C07305=1237.701,70.398,-44.996,-178.646,5.352,148.520
C07306=1237.696,70.648,-45.014,-178.643,5.352,148.519
C07307=1237.691,70.897,-45.032,-178.640,5.353,148.519
C07308=1237.686,71.147,-45.049,-178.638,5.353,148.518
C07309=1237.681,71.396,-45.067,-178.635,5.354,148.517
C07310=1237.677,71.645,-45.084,-178.633,5.355,148.517
C07311=1237.671,71.894,-45.102,-178.630,5.355,148.516
C07312=1237.666,72.144,-45.120,-178.628,5.356,148.516
C07313=1237.662,72.393,-45.137,-178.625,5.357,148.515
C07314=1237.656,72.643,-45.155,-178.623,5.357,148.514
C07315=1237.652,72.891,-45.172,-178.620,5.358,148.514
C07316=1237.647,73.141,-45.190,-178.618,5.358,148.513
C07317=1237.642,73.390,-45.208,-178.615,5.358,148.512
C07318=1237.637,73.640,-45.225,-178.613,5.359,148.512
C07319=1237.632,73.889,-45.243,-178.610,5.360,148.511
C07320=1237.627,74.138,-45.261,-178.608,5.360,148.511
C07321=1237.622,74.387,-45.279,-178.605,5.361,148.510
C07322=1237.617,74.637,-45.297,-178.603,5.362,148.509
C07323=1237.613,74.886,-45.314,-178.600,5.362,148.509
C07324=1237.608,75.135,-45.332,-178.597,5.363,148.508
C07325=1237.603,75.384,-45.350,-178.595,5.364,148.508
C07326=1237.599,75.635,-45.368,-178.593,5.364,148.507
C07327=1237.594,75.884,-45.386,-178.590,5.365,148.506
C07328=1237.589,76.133,-45.403,-178.587,5.366,148.506
C07329=1237.584,76.382,-45.421,-178.585,5.366,148.505
C07330=1237.579,76.631,-45.439,-178.582,5.367,148.504
C07331=1237.574,76.880,-45.457,-178.579,5.367,148.504
C07332=1237.569,77.130,-45.475,-178.577,5.368,148.503
C07333=1237.564,77.379,-45.493,-178.575,5.369,148.503
C07334=1237.559,77.629,-45.511,-178.572,5.370,148.502
C07335=1237.555,77.878,-45.528,-178.569,5.370,148.501
C07336=1237.550,78.127,-45.546,-178.567,5.371,148.501
C07337=1237.545,78.376,-45.564,-178.564,5.371,148.500
C07338=1237.541,78.626,-45.582,-178.562,5.372,148.499
C07339=1237.536,78.875,-45.600,-178.559,5.373,148.499
C07340=1237.531,79.125,-45.618,-178.557,5.374,148.498
C07341=1237.526,79.374,-45.636,-178.554,5.374,148.498
C07342=1237.521,79.623,-45.654,-178.552,5.375,148.497
C07343=1237.516,79.872,-45.672,-178.549,5.376,148.496
C07344=1237.511,80.121,-45.690,-178.547,5.376,148.496
C07345=1237.506,80.371,-45.707,-178.544,5.377,148.495
C07346=1237.502,80.620,-45.726,-178.542,5.378,148.494
C07347=1237.497,80.870,-45.744,-178.539,5.378,148.494
C07348=1237.492,81.119,-45.762,-178.536,5.379,148.493
C07349=1237.486,81.368,-45.780,-178.534,5.380,148.493
C07350=1237.481,81.637,-45.800,-178.532,5.380,148.492
C07351=1237.476,81.905,-45.819,-178.529,5.381,148.491
C07352=1237.471,82.173,-45.839,-178.526,5.382,148.491
C07353=1237.466,82.441,-45.858,-178.523,5.383,148.490
C07354=1237.461,82.690,-45.876,-178.520,5.384,148.489
C07355=1237.457,82.940,-45.894,-178.518,5.384,148.489
C07356=1237.452,83.190,-45.912,-178.515,5.385,148.488
C07357=1237.446,83.439,-45.931,-178.513,5.385,148.487
C07358=1237.441,83.688,-45.949,-178.510,5.386,148.487
C07359=1237.436,83.937,-45.967,-178.508,5.387,148.486
C07360=1237.431,84.187,-45.985,-178.505,5.388,148.486
C07361=1237.427,84.436,-46.003,-178.503,5.388,148.485
C07362=1237.422,84.686,-46.021,-178.500,5.389,148.484
C07363=1237.417,84.935,-46.039,-178.497,5.389,148.484
C07364=1237.413,85.183,-46.058,-178.495,5.390,148.483
C07365=1237.408,85.433,-46.076,-178.493,5.391,148.483
C07366=1237.403,85.683,-46.095,-178.490,5.392,148.482
C07367=1237.398,85.932,-46.113,-178.487,5.392,148.481
C07368=1237.393,86.181,-46.131,-178.485,5.393,148.481
C07369=1237.388,86.430,-46.149,-178.483,5.394,148.480
C07370=1237.384,86.680,-46.167,-178.480,5.394,148.480
C07371=1237.379,86.929,-46.186,-178.477,5.395,148.479
C07372=1237.373,87.178,-46.204,-178.475,5.396,148.478
C07373=1237.368,87.427,-46.222,-178.472,5.396,148.478
C07374=1237.364,87.677,-46.241,-178.470,5.397,148.477
C07375=1237.359,87.926,-46.259,-178.467,5.398,148.477
C07376=1237.355,88.175,-46.277,-178.465,5.398,148.476
C07377=1237.349,88.424,-46.296,-178.462,5.399,148.475
C07378=1237.345,88.674,-46.314,-178.460,5.400,148.475
C07379=1237.340,88.923,-46.332,-178.457,5.401,148.474
C07380=1237.335,89.172,-46.351,-178.455,5.401,148.474
C07381=1237.330,89.421,-46.369,-178.452,5.402,148.473
C07382=1237.325,89.671,-46.388,-178.449,5.402,148.472
C07383=1237.320,89.921,-46.406,-178.447,5.403,148.472
C07384=1237.316,90.169,-46.424,-178.445,5.404,148.471
C07385=1237.311,90.419,-46.443,-178.442,5.405,148.471
C07386=1237.306,90.668,-46.461,-178.439,5.405,148.470
C07387=1237.301,90.917,-46.480,-178.437,5.406,148.469
C07388=1237.296,91.166,-46.498,-178.434,5.408,148.469
C07389=1237.291,91.416,-46.517,-178.432,5.408,148.468
C07390=1237.286,91.665,-46.536,-178.429,5.409,148.468
C07391=1237.282,91.914,-46.554,-178.426,5.409,148.467
C07392=1237.277,92.164,-46.572,-178.424,5.410,148.466
C07393=1237.272,92.413,-46.591,-178.422,5.411,148.466
C07394=1237.267,92.662,-46.609,-178.419,5.412,148.465
C07395=1237.263,92.911,-46.628,-178.416,5.412,148.465
C07396=1237.257,93.161,-46.647,-178.414,5.413,148.464
C07397=1237.252,93.410,-46.665,-178.412,5.414,148.463
C07398=1237.248,93.659,-46.684,-178.409,5.414,148.463
C07399=1237.243,93.909,-46.703,-178.406,5.415,148.462
C07400=1237.238,94.157,-46.721,-178.404,5.416,148.461
C07401=1237.234,94.407,-46.740,-178.402,5.417,148.461
C07402=1237.229,94.656,-46.759,-178.399,5.417,148.460
C07403=1237.224,94.905,-46.777,-178.396,5.418,148.460
C07404=1237.219,95.155,-46.795,-178.393,5.419,148.459
C07405=1237.214,95.404,-46.815,-178.391,5.420,148.459
C07406=1237.209,95.653,-46.833,-178.388,5.421,148.458
C07407=1237.204,95.903,-46.852,-178.386,5.422,148.457
C07408=1237.199,96.152,-46.870,-178.383,5.422,148.457
C07409=1237.195,96.401,-46.889,-178.381,5.423,148.456
C07410=1237.190,96.651,-46.908,-178.378,5.424,148.456
C07411=1237.185,96.899,-46.926,-178.376,5.424,148.455
C07412=1237.180,97.149,-46.946,-178.373,5.425,148.454
C07413=1237.175,97.398,-46.964,-178.371,5.426,148.454
C07414=1237.171,97.647,-46.984,-178.368,5.427,148.453
C07415=1237.166,97.897,-47.002,-178.366,5.427,148.453
C07416=1237.161,98.145,-47.020,-178.363,5.428,148.452
C07417=1237.156,98.395,-47.039,-178.361,5.430,148.452
C07418=1237.152,98.644,-47.058,-178.358,5.430,148.451
C07419=1237.147,98.894,-47.078,-178.355,5.431,148.450
C07420=1237.142,99.143,-47.096,-178.353,5.432,148.450
C07421=1237.137,99.392,-47.115,-178.351,5.432,148.449
C07422=1237.132,99.641,-47.133,-178.348,5.433,148.449
C07423=1237.127,99.890,-47.153,-178.345,5.434,148.448
C07424=1237.123,100.140,-47.172,-178.343,5.435,148.448
C07425=1237.117,100.389,-47.190,-178.341,5.435,148.447
C07426=1237.113,100.638,-47.209,-178.338,5.436,148.446
C07427=1237.108,100.887,-47.229,-178.335,5.437,148.446
C07428=1237.104,101.137,-47.247,-178.333,5.438,148.445
C07429=1237.098,101.386,-47.266,-178.330,5.439,148.445
C07430=1237.094,101.635,-47.285,-178.327,5.440,148.444
C07431=1237.089,101.885,-47.304,-178.325,5.440,148.443
C07432=1237.084,102.133,-47.323,-178.323,5.441,148.443
C07433=1237.079,102.383,-47.342,-178.320,5.442,148.442
C07434=1237.075,102.631,-47.361,-178.317,5.442,148.442
C07435=1237.070,102.882,-47.380,-178.315,5.443,148.441
C07436=1237.065,103.130,-47.399,-178.313,5.444,148.440
C07437=1237.060,103.380,-47.418,-178.310,5.445,148.440
C07438=1237.055,103.629,-47.438,-178.307,5.446,148.439
C07439=1237.051,103.878,-47.456,-178.305,5.447,148.439
C07440=1237.045,104.127,-47.475,-178.302,5.448,148.438
C07441=1237.041,104.377,-47.494,-178.300,5.448,148.437
C07442=1237.036,104.625,-47.514,-178.297,5.449,148.437
C07443=1237.031,104.876,-47.532,-178.295,5.450,148.436
C07444=1237.026,105.124,-47.551,-178.292,5.451,148.436
C07445=1237.021,105.374,-47.571,-178.290,5.451,148.435
C07446=1237.017,105.622,-47.590,-178.287,5.453,148.435
C07447=1237.012,105.872,-47.609,-178.284,5.454,148.434
C07448=1237.007,106.121,-47.628,-178.282,5.454,148.433
C07449=1237.003,106.370,-47.648,-178.280,5.455,148.433
C07450=1236.998,106.620,-47.666,-178.277,5.456,148.432
C07451=1236.992,106.869,-47.686,-178.274,5.456,148.432
C07452=1236.988,107.118,-47.705,-178.272,5.457,148.431
C07453=1236.983,107.367,-47.724,-178.270,5.458,148.431
C07454=1236.978,107.636,-47.745,-178.266,5.459,148.430
C07455=1236.973,107.904,-47.766,-178.264,5.460,148.429
C07456=1236.967,108.173,-47.786,-178.261,5.461,148.429
C07457=1236.962,108.442,-47.807,-178.258,5.462,148.428
C07458=1236.958,108.690,-47.826,-178.256,5.463,148.428
C07459=1236.953,108.940,-47.846,-178.253,5.464,148.427
C07460=1236.948,109.189,-47.865,-178.251,5.464,148.426
C07461=1236.943,109.438,-47.885,-178.248,5.465,148.426
C07462=1236.938,109.687,-47.903,-178.246,5.466,148.425
C07463=1236.934,109.936,-47.923,-178.243,5.467,148.425
C07464=1236.929,110.186,-47.943,-178.240,5.468,148.424
C07465=1236.924,110.434,-47.961,-178.238,5.469,148.424
C07466=1236.920,110.684,-47.981,-178.235,5.470,148.423
C07467=1236.914,110.933,-48.000,-178.233,5.470,148.422
C07468=1236.910,111.182,-48.020,-178.231,5.471,148.422
C07469=1236.905,111.432,-48.040,-178.228,5.472,148.421
C07470=1236.900,111.681,-48.058,-178.225,5.473,148.421
C07471=1236.895,111.930,-48.078,-178.223,5.474,148.420
C07472=1236.891,112.180,-48.098,-178.220,5.475,148.420
C07473=1236.885,112.429,-48.117,-178.218,5.476,148.419
C07474=1236.881,112.678,-48.136,-178.215,5.477,148.419
C07475=1236.876,112.926,-48.156,-178.213,5.477,148.418
C07476=1236.872,113.176,-48.176,-178.210,5.479,148.417
C07477=1236.867,113.425,-48.195,-178.208,5.480,148.417
C07478=1236.861,113.674,-48.215,-178.205,5.480,148.416
C07479=1236.857,113.924,-48.234,-178.202,5.481,148.416
C07480=1236.853,114.173,-48.253,-178.200,5.482,148.415
C07481=1236.847,114.422,-48.273,-178.198,5.483,148.415
C07482=1236.843,114.671,-48.292,-178.194,5.484,148.414
C07483=1236.838,114.920,-48.313,-178.192,5.485,148.414
C07484=1236.833,115.169,-48.332,-178.190,5.486,148.413
C07485=1236.828,115.419,-48.352,-178.187,5.486,148.412
C07486=1236.823,115.668,-48.371,-178.185,5.487,148.412
C07487=1236.819,115.917,-48.390,-178.182,5.488,148.411
C07488=1236.814,116.166,-48.410,-178.179,5.489,148.411
C07489=1236.810,116.415,-48.430,-178.177,5.490,148.410
C07490=1236.804,116.664,-48.449,-178.174,5.491,148.410
C07491=1236.799,116.914,-48.469,-178.172,5.492,148.409
C07492=1236.795,117.163,-48.489,-178.170,5.493,148.408
C07493=1236.790,117.412,-48.509,-178.167,5.494,148.408
C07494=1236.785,117.661,-48.528,-178.164,5.495,148.407
C07495=1236.780,117.911,-48.548,-178.162,5.496,148.407
C07496=1236.776,118.160,-48.568,-178.159,5.496,148.406
C07497=1236.770,118.409,-48.588,-178.157,5.497,148.406
C07498=1236.766,118.658,-48.607,-178.154,5.499,148.405
C07499=1236.762,118.907,-48.627,-178.151,5.499,148.405
C07500=1236.757,119.156,-48.647,-178.149,5.500,148.404
C07501=1236.752,119.405,-48.666,-178.147,5.501,148.403
C07502=1236.747,119.654,-48.686,-178.144,5.502,148.403
C07503=1236.743,119.904,-48.706,-178.142,5.503,148.402
C07504=1236.738,120.153,-48.726,-178.139,5.504,148.402
C07505=1236.733,120.402,-48.746,-178.136,5.505,148.401
C07506=1236.728,120.651,-48.765,-178.134,5.506,148.401
C07507=1236.723,120.901,-48.785,-178.131,5.506,148.400
C07508=1236.719,121.150,-48.805,-178.128,5.508,148.399
C07509=1236.714,121.399,-48.825,-178.126,5.509,148.399
C07510=1236.709,121.647,-48.845,-178.123,5.509,148.398
C07511=1236.704,121.897,-48.865,-178.121,5.510,148.398
C07512=1236.700,122.147,-48.884,-178.119,5.511,148.397
C07513=1236.695,122.396,-48.905,-178.116,5.513,148.397
C07514=1236.689,122.645,-48.925,-178.113,5.513,148.396
C07515=1236.685,122.894,-48.945,-178.111,5.514,148.396
C07516=1236.680,123.143,-48.965,-178.109,5.515,148.395
C07517=1236.676,123.392,-48.985,-178.106,5.516,148.395
C07518=1236.671,123.642,-49.005,-178.103,5.517,148.394
C07519=1236.666,123.890,-49.025,-178.101,5.518,148.394
C07520=1236.661,124.140,-49.044,-178.098,5.519,148.393
C07521=1236.657,124.389,-49.065,-178.096,5.519,148.392
C07522=1236.652,124.638,-49.084,-178.093,5.521,148.392
C07523=1236.647,124.887,-49.105,-178.090,5.522,148.391
C07524=1236.643,125.137,-49.124,-178.088,5.523,148.391
C07525=1236.638,125.385,-49.144,-178.086,5.524,148.390
C07526=1236.632,125.635,-49.165,-178.083,5.524,148.390
C07527=1236.628,125.884,-49.185,-178.080,5.526,148.389
C07528=1236.623,126.133,-49.205,-178.078,5.527,148.389
C07529=1236.619,126.382,-49.225,-178.076,5.528,148.388
C07530=1236.614,126.631,-49.245,-178.073,5.528,148.388
C07531=1236.609,126.880,-49.265,-178.070,5.530,148.387
C07532=1236.604,127.129,-49.285,-178.068,5.531,148.387
C07533=1236.599,127.378,-49.306,-178.065,5.531,148.386
C07534=1236.594,127.628,-49.326,-178.063,5.532,148.386
C07535=1236.590,127.877,-49.346,-178.060,5.534,148.385
C07536=1236.585,128.126,-49.366,-178.057,5.534,148.384
C07537=1236.581,128.375,-49.386,-178.055,5.535,148.384
C07538=1236.576,128.624,-49.406,-178.053,5.536,148.383
C07539=1236.571,128.874,-49.427,-178.050,5.538,148.383
C07540=1236.566,129.122,-49.447,-178.047,5.539,148.382
C07541=1236.561,129.371,-49.467,-178.045,5.539,148.382
C07542=1236.557,129.620,-49.487,-178.043,5.540,148.381
C07543=1236.552,129.870,-49.508,-178.039,5.542,148.381
C07544=1236.547,130.119,-49.528,-178.037,5.543,148.380
C07545=1236.543,130.368,-49.548,-178.035,5.543,148.380
C07546=1236.538,130.618,-49.568,-178.033,5.544,148.379
C07547=1236.533,130.867,-49.588,-178.029,5.546,148.379
C07548=1236.528,131.116,-49.609,-178.027,5.546,148.378
C07549=1236.524,131.365,-49.630,-178.025,5.547,148.377
C07550=1236.519,131.614,-49.650,-178.022,5.548,148.377
C07551=1236.514,131.864,-49.670,-178.019,5.550,148.376
C07552=1236.509,132.112,-49.690,-178.017,5.551,148.376
C07553=1236.504,132.361,-49.711,-178.015,5.552,148.375
C07554=1236.500,132.610,-49.731,-178.012,5.553,148.375
C07555=1236.495,132.859,-49.752,-178.009,5.554,148.374
C07556=1236.490,133.109,-49.772,-178.007,5.555,148.374
C07557=1236.486,133.357,-49.792,-178.004,5.555,148.373
C07558=1236.480,133.626,-49.815,-178.001,5.557,148.373
C07559=1236.475,133.896,-49.837,-177.999,5.558,148.372
C07560=1236.470,134.164,-49.859,-177.996,5.559,148.372
C07561=1236.465,134.432,-49.881,-177.993,5.560,148.371
C07562=1236.460,134.681,-49.902,-177.991,5.561,148.370
C07563=1236.455,134.931,-49.921,-177.988,5.562,148.370
C07564=1236.451,135.180,-49.942,-177.986,5.563,148.369
C07565=1236.446,135.429,-49.963,-177.983,5.564,148.369
C07566=1236.441,135.678,-49.983,-177.980,5.565,148.368
C07567=1236.436,135.927,-50.004,-177.978,5.566,148.368
C07568=1236.432,136.176,-50.024,-177.975,5.567,148.367
C07569=1236.427,136.425,-50.045,-177.973,5.568,148.367
C07570=1236.422,136.674,-50.066,-177.970,5.570,148.366
C07571=1236.418,136.923,-50.086,-177.968,5.571,148.366
C07572=1236.413,137.172,-50.107,-177.965,5.571,148.365
C07573=1236.408,137.421,-50.127,-177.963,5.573,148.365
C07574=1236.404,137.670,-50.148,-177.960,5.574,148.364
C07575=1236.398,137.920,-50.169,-177.958,5.575,148.364
C07576=1236.395,138.169,-50.190,-177.955,5.576,148.363
C07577=1236.389,138.419,-50.211,-177.952,5.577,148.363
C07578=1236.385,138.668,-50.231,-177.950,5.578,148.362
C07579=1236.380,138.917,-50.252,-177.948,5.578,148.361
C07580=1236.375,139.166,-50.272,-177.945,5.580,148.361
C07581=1236.370,139.415,-50.293,-177.942,5.581,148.360
C07582=1236.366,139.664,-50.314,-177.940,5.582,148.360
C07583=1236.361,139.913,-50.335,-177.937,5.583,148.359
C07584=1236.356,140.162,-50.356,-177.935,5.584,148.359
C07585=1236.351,140.411,-50.377,-177.932,5.585,148.358
C07586=1236.347,140.660,-50.397,-177.930,5.587,148.358
C07587=1236.342,140.909,-50.418,-177.927,5.588,148.357
C07588=1236.337,141.158,-50.438,-177.925,5.589,148.357
C07589=1236.332,141.407,-50.459,-177.922,5.590,148.356
C07590=1236.328,141.656,-50.480,-177.920,5.591,148.356
C07591=1236.323,141.906,-50.501,-177.917,5.592,148.355
C07592=1236.319,142.154,-50.522,-177.914,5.593,148.355
C07593=1236.314,142.404,-50.543,-177.912,5.594,148.354
C07594=1236.309,142.653,-50.563,-177.910,5.595,148.354
C07595=1236.304,142.902,-50.584,-177.907,5.597,148.353
C07596=1236.300,143.151,-50.605,-177.904,5.598,148.353
C07597=1236.295,143.399,-50.626,-177.902,5.598,148.352
C07598=1236.290,143.649,-50.647,-177.899,5.600,148.352
C07599=1236.286,143.898,-50.668,-177.897,5.601,148.351
C07600=1236.281,144.148,-50.689,-177.894,5.601,148.351
C07601=1236.277,144.396,-50.710,-177.891,5.603,148.350
C07602=1236.271,144.645,-50.731,-177.889,5.604,148.350
C07603=1236.266,144.894,-50.752,-177.887,5.605,148.349
C07604=1236.262,145.143,-50.772,-177.883,5.606,148.349
C07605=1236.257,145.392,-50.794,-177.881,5.607,148.348
C07606=1236.253,145.642,-50.815,-177.879,5.608,148.348
C07607=1236.248,145.891,-50.836,-177.876,5.610,148.347
C07608=1236.243,146.140,-50.858,-177.874,5.611,148.347
C07609=1236.239,146.389,-50.878,-177.871,5.612,148.346
C07610=1236.233,146.638,-50.899,-177.868,5.613,148.346
C07611=1236.229,146.886,-50.921,-177.866,5.614,148.345
C07612=1236.225,147.136,-50.941,-177.864,5.615,148.345
C07613=1236.220,147.385,-50.962,-177.861,5.616,148.344
C07614=1236.215,147.634,-50.984,-177.859,5.617,148.344
C07615=1236.210,147.883,-51.004,-177.856,5.618,148.343
C07616=1236.205,148.132,-51.026,-177.854,5.620,148.343
C07617=1236.201,148.382,-51.047,-177.851,5.621,148.342
C07618=1236.196,148.631,-51.068,-177.848,5.622,148.342
C07619=1236.191,148.879,-51.089,-177.846,5.623,148.341
C07620=1236.186,149.128,-51.110,-177.844,5.624,148.341
C07621=1236.182,149.378,-51.132,-177.840,5.626,148.340
C07622=1236.178,149.627,-51.153,-177.838,5.627,148.340
C07623=1236.173,149.875,-51.174,-177.836,5.627,148.339
C07624=1236.168,150.125,-51.195,-177.833,5.629,148.339
C07625=1236.163,150.373,-51.217,-177.830,5.630,148.338
C07626=1236.159,150.623,-51.238,-177.828,5.632,148.338
C07627=1236.154,150.872,-51.260,-177.825,5.632,148.337
C07628=1236.149,151.121,-51.281,-177.823,5.633,148.337
C07629=1236.144,151.369,-51.302,-177.820,5.635,148.336
C07630=1236.140,151.619,-51.323,-177.818,5.636,148.336
C07631=1236.135,151.868,-51.345,-177.815,5.636,148.335
C07632=1236.130,152.117,-51.366,-177.813,5.638,148.335
C07633=1236.125,152.366,-51.387,-177.811,5.639,148.334
C07634=1236.121,152.616,-51.409,-177.807,5.641,148.334
C07635=1236.116,152.864,-51.430,-177.805,5.642,148.333
C07636=1236.111,153.113,-51.451,-177.803,5.642,148.333
C07637=1236.107,153.363,-51.473,-177.800,5.644,148.332
C07638=1236.102,153.611,-51.494,-177.797,5.645,148.332
C07639=1236.097,153.860,-51.515,-177.795,5.647,148.332
C07640=1236.092,154.109,-51.537,-177.792,5.647,148.331
C07641=1236.088,154.359,-51.558,-177.790,5.648,148.330
C07642=1236.083,154.607,-51.579,-177.787,5.650,148.330
C07643=1236.079,154.856,-51.601,-177.785,5.651,148.329
C07644=1236.074,155.106,-51.622,-177.782,5.653,148.329
C07645=1236.069,155.355,-51.644,-177.780,5.653,148.328
C07646=1236.064,155.603,-51.666,-177.777,5.654,148.328
C07647=1236.060,155.853,-51.687,-177.774,5.656,148.328
C07648=1236.055,156.102,-51.709,-177.772,5.657,148.327
C07649=1236.050,156.350,-51.731,-177.769,5.658,148.327
C07650=1236.046,156.600,-51.753,-177.767,5.659,148.326
C07651=1236.041,156.849,-51.773,-177.765,5.660,148.326
C07652=1236.036,157.097,-51.795,-177.762,5.662,148.325
C07653=1236.032,157.347,-51.817,-177.760,5.663,148.325
C07654=1236.027,157.595,-51.838,-177.756,5.664,148.324
C07655=1236.022,157.845,-51.859,-177.754,5.665,148.324
C07656=1236.018,158.094,-51.881,-177.752,5.666,148.323
C07657=1236.013,158.343,-51.903,-177.749,5.668,148.323
C07658=1236.009,158.592,-51.925,-177.747,5.669,148.322
C07659=1236.004,158.841,-51.947,-177.744,5.670,148.322
C07660=1235.999,159.090,-51.968,-177.742,5.671,148.321
C07661=1235.994,159.339,-51.990,-177.739,5.673,148.321
C07662=1235.989,159.608,-52.014,-177.737,5.674,148.320
C07663=1235.984,159.877,-52.037,-177.733,5.675,148.320
C07664=1235.979,160.146,-52.060,-177.731,5.676,148.319
C07665=1235.974,160.415,-52.084,-177.728,5.678,148.319
C07666=1235.969,160.664,-52.106,-177.725,5.679,148.318
C07667=1235.964,160.914,-52.127,-177.723,5.680,148.318
C07668=1235.959,161.162,-52.149,-177.721,5.681,148.317
C07669=1235.955,161.412,-52.171,-177.718,5.683,148.317
C07670=1235.950,161.660,-52.193,-177.716,5.684,148.316
C07671=1235.946,161.910,-52.215,-177.712,5.685,148.316
C07672=1235.941,162.158,-52.236,-177.710,5.686,148.315
C07673=1235.936,162.407,-52.258,-177.708,5.688,148.315
C07674=1235.932,162.656,-52.280,-177.705,5.689,148.315
C07675=1235.927,162.905,-52.302,-177.702,5.691,148.314
C07676=1235.923,163.154,-52.324,-177.700,5.691,148.314
C07677=1235.918,163.403,-52.345,-177.698,5.692,148.313
C07678=1235.913,163.653,-52.368,-177.695,5.694,148.313
C07679=1235.908,163.901,-52.390,-177.692,5.695,148.312
C07680=1235.904,164.151,-52.412,-177.690,5.697,148.312
C07681=1235.899,164.399,-52.433,-177.687,5.697,148.311
C07682=1235.895,164.649,-52.455,-177.685,5.699,148.311
C07683=1235.890,164.897,-52.477,-177.682,5.700,148.310
C07684=1235.886,165.147,-52.499,-177.679,5.702,148.310
C07685=1235.881,165.395,-52.521,-177.677,5.703,148.309
C07686=1235.876,165.645,-52.544,-177.674,5.704,148.309
C07687=1235.871,165.893,-52.565,-177.672,5.705,148.308
C07688=1235.867,166.143,-52.587,-177.669,5.707,148.308
C07689=1235.862,166.391,-52.609,-177.667,5.708,148.307
C07690=1235.858,166.640,-52.632,-177.665,5.709,148.307
C07691=1235.853,166.889,-52.653,-177.662,5.711,148.307
C07692=1235.848,167.138,-52.676,-177.659,5.711,148.306
C07693=1235.843,167.387,-52.698,-177.657,5.713,148.306
C07694=1235.839,167.636,-52.720,-177.654,5.714,148.305
C07695=1235.834,167.885,-52.741,-177.652,5.716,148.305
C07696=1235.830,168.134,-52.764,-177.649,5.717,148.304
C07697=1235.824,168.383,-52.786,-177.646,5.718,148.304
C07698=1235.820,168.632,-52.809,-177.644,5.719,148.303
C07699=1235.815,168.881,-52.830,-177.642,5.721,148.303
C07700=1235.811,169.130,-52.852,-177.639,5.722,148.302
C07701=1235.805,169.379,-52.875,-177.636,5.724,148.302
C07702=1235.801,169.628,-52.897,-177.634,5.725,148.302
C07703=1235.796,169.876,-52.919,-177.631,5.726,148.301
C07704=1235.792,170.126,-52.941,-177.629,5.727,148.301
C07705=1235.787,170.375,-52.964,-177.626,5.729,148.300
C07706=1235.783,170.623,-52.986,-177.624,5.730,148.300
C07707=1235.778,170.873,-53.008,-177.621,5.732,148.299
C07708=1235.773,171.122,-53.030,-177.619,5.732,148.299
C07709=1235.768,171.371,-53.052,-177.616,5.734,148.298
C07710=1235.764,171.619,-53.075,-177.614,5.735,148.298
C07711=1235.760,171.868,-53.097,-177.611,5.737,148.297
C07712=1235.755,172.118,-53.120,-177.609,5.738,148.297
C07713=1235.750,172.366,-53.142,-177.606,5.739,148.297
C07714=1235.746,172.615,-53.164,-177.603,5.740,148.296
C07715=1235.740,172.864,-53.186,-177.601,5.742,148.296
C07716=1235.736,173.113,-53.209,-177.599,5.743,148.295
C07717=1235.731,173.363,-53.232,-177.595,5.744,148.295
C07718=1235.727,173.611,-53.254,-177.593,5.745,148.294
C07719=1235.722,173.860,-53.276,-177.591,5.747,148.294
C07720=1235.717,174.110,-53.299,-177.588,5.748,148.293
C07721=1235.713,174.358,-53.321,-177.585,5.750,148.293
C07722=1235.709,174.607,-53.343,-177.583,5.751,148.293
C07723=1235.703,174.855,-53.366,-177.580,5.752,148.292
C07724=1235.699,175.105,-53.388,-177.578,5.753,148.292
C07725=1235.694,175.354,-53.411,-177.576,5.755,148.291
C07726=1235.689,175.602,-53.433,-177.573,5.756,148.291
C07727=1235.685,175.852,-53.455,-177.570,5.758,148.290
C07728=1235.680,176.101,-53.479,-177.568,5.760,148.290
C07729=1235.676,176.349,-53.500,-177.565,5.760,148.289
C07730=1235.671,176.598,-53.524,-177.562,5.762,148.289
C07731=1235.667,176.848,-53.546,-177.560,5.763,148.289
C07732=1235.661,177.096,-53.569,-177.557,5.765,148.288
C07733=1235.657,177.346,-53.591,-177.555,5.766,148.288
C07734=1235.652,177.595,-53.614,-177.552,5.768,148.287
C07735=1235.648,177.843,-53.637,-177.550,5.769,148.287
C07736=1235.643,178.092,-53.659,-177.547,5.770,148.286
C07737=1235.639,178.341,-53.682,-177.545,5.771,148.286
C07738=1235.634,178.591,-53.705,-177.542,5.773,148.286
C07739=1235.629,178.839,-53.727,-177.540,5.774,148.285
C07740=1235.624,179.088,-53.750,-177.537,5.775,148.285
C07741=1235.620,179.337,-53.772,-177.535,5.777,148.284
C07742=1235.615,179.585,-53.795,-177.532,5.778,148.284
C07743=1235.611,179.835,-53.817,-177.529,5.780,148.283
C07744=1235.606,180.084,-53.841,-177.527,5.781,148.283
C07745=1235.602,180.332,-53.864,-177.524,5.782,148.282
C07746=1235.596,180.581,-53.886,-177.522,5.783,148.282
C07747=1235.592,180.830,-53.909,-177.519,5.785,148.282
C07748=1235.588,181.079,-53.932,-177.517,5.786,148.281
C07749=1235.583,181.329,-53.955,-177.514,5.788,148.281
C07750=1235.578,181.577,-53.977,-177.512,5.790,148.280
C07751=1235.574,181.826,-54.000,-177.509,5.791,148.280
C07752=1235.569,182.075,-54.022,-177.506,5.792,148.279
C07753=1235.565,182.324,-54.046,-177.504,5.793,148.279
C07754=1235.560,182.572,-54.068,-177.502,5.795,148.279
C07755=1235.555,182.821,-54.092,-177.500,5.796,148.278
C07756=1235.550,183.071,-54.114,-177.496,5.798,148.278
C07757=1235.546,183.320,-54.137,-177.494,5.799,148.277
C07758=1235.542,183.569,-54.160,-177.492,5.800,148.277
C07759=1235.536,183.817,-54.183,-177.489,5.802,148.276
C07760=1235.532,184.066,-54.206,-177.486,5.803,148.276
C07761=1235.527,184.315,-54.229,-177.484,5.805,148.276
C07762=1235.523,184.564,-54.252,-177.481,5.807,148.275
C07763=1235.519,184.813,-54.275,-177.479,5.807,148.275
C07764=1235.513,185.061,-54.298,-177.476,5.809,148.274
C07765=1235.509,185.310,-54.321,-177.474,5.810,148.274
C07766=1235.504,185.580,-54.346,-177.471,5.812,148.273
C07767=1235.499,185.850,-54.371,-177.468,5.814,148.273
C07768=1235.494,186.120,-54.396,-177.465,5.815,148.272
C07769=1235.489,186.390,-54.421,-177.462,5.817,148.272
C07770=1235.484,186.638,-54.444,-177.460,5.818,148.272
C07771=1235.479,186.887,-54.467,-177.458,5.820,148.271
C07772=1235.476,187.136,-54.490,-177.455,5.821,148.271
C07773=1235.471,187.385,-54.513,-177.452,5.822,148.270
C07774=1235.466,187.634,-54.536,-177.450,5.824,148.270
C07775=1235.461,187.883,-54.560,-177.447,5.825,148.270
C07776=1235.457,188.132,-54.582,-177.445,5.827,148.269
C07777=1235.452,188.380,-54.605,-177.442,5.828,148.269
C07778=1235.447,188.629,-54.629,-177.440,5.830,148.268
C07779=1235.443,188.878,-54.652,-177.437,5.832,148.268
C07780=1235.439,189.127,-54.675,-177.435,5.832,148.267
C07781=1235.434,189.376,-54.698,-177.432,5.834,148.267
C07782=1235.429,189.625,-54.722,-177.430,5.835,148.267
C07783=1235.425,189.874,-54.745,-177.427,5.837,148.266
C07784=1235.420,190.123,-54.768,-177.424,5.838,148.266
C07785=1235.415,190.372,-54.792,-177.422,5.839,148.265
C07786=1235.411,190.620,-54.814,-177.419,5.841,148.265
C07787=1235.406,190.869,-54.838,-177.417,5.843,148.265
C07788=1235.401,191.118,-54.861,-177.414,5.844,148.264
C07789=1235.397,191.367,-54.884,-177.412,5.846,148.264
C07790=1235.392,191.616,-54.908,-177.409,5.847,148.263
C07791=1235.387,191.865,-54.931,-177.407,5.849,148.263
C07792=1235.383,192.114,-54.954,-177.404,5.850,148.263
C07793=1235.379,192.362,-54.978,-177.402,5.851,148.262
C07794=1235.374,192.611,-55.001,-177.399,5.853,148.262
C07795=1235.369,192.860,-55.025,-177.396,5.855,148.261
C07796=1235.365,193.109,-55.048,-177.394,5.856,148.261
C07797=1235.360,193.358,-55.071,-177.391,5.857,148.261
C07798=1235.355,193.607,-55.095,-177.389,5.858,148.260
C07799=1235.351,193.856,-55.119,-177.386,5.860,148.260
C07800=1235.346,194.105,-55.142,-177.384,5.862,148.259
C07801=1235.342,194.354,-55.165,-177.381,5.863,148.259
C07802=1235.337,194.603,-55.189,-177.379,5.865,148.258
C07803=1235.332,194.851,-55.211,-177.376,5.867,148.258
C07804=1235.328,195.099,-55.235,-177.374,5.868,148.258
C07805=1235.323,195.348,-55.259,-177.371,5.869,148.257
C07806=1235.319,195.597,-55.282,-177.368,5.871,148.257
C07807=1235.314,195.846,-55.305,-177.366,5.872,148.256
C07808=1235.309,196.095,-55.329,-177.363,5.874,148.256
C07809=1235.305,196.344,-55.353,-177.361,5.876,148.256
C07810=1235.300,196.593,-55.376,-177.359,5.877,148.255
C07811=1235.296,196.841,-55.400,-177.355,5.878,148.255
C07812=1235.291,197.090,-55.424,-177.353,5.880,148.255
C07813=1235.287,197.340,-55.447,-177.351,5.881,148.254
C07814=1235.282,197.588,-55.471,-177.348,5.883,148.254
C07815=1235.278,197.837,-55.495,-177.345,5.885,148.253
C07816=1235.273,198.086,-55.518,-177.343,5.886,148.253
C07817=1235.269,198.335,-55.542,-177.340,5.887,148.253
C07818=1235.264,198.584,-55.565,-177.338,5.889,148.252
C07819=1235.260,198.832,-55.590,-177.336,5.890,148.252
C07820=1235.255,199.081,-55.613,-177.333,5.892,148.251
C07821=1235.249,199.331,-55.637,-177.330,5.894,148.251
C07822=1235.245,199.579,-55.661,-177.328,5.895,148.251
C07823=1235.240,199.828,-55.684,-177.325,5.897,148.250
C07824=1235.236,200.077,-55.708,-177.322,5.898,148.250
C07825=1235.231,200.326,-55.732,-177.320,5.900,148.249
C07826=1235.227,200.574,-55.756,-177.318,5.901,148.249
C07827=1235.222,200.823,-55.779,-177.315,5.903,148.249
C07828=1235.218,201.071,-55.803,-177.312,5.905,148.248
C07829=1235.213,201.320,-55.827,-177.310,5.906,148.248
C07830=1235.209,201.570,-55.851,-177.307,5.908,148.248
C07831=1235.204,201.819,-55.875,-177.305,5.910,148.247
C07832=1235.199,202.067,-55.899,-177.303,5.911,148.247
C07833=1235.195,202.316,-55.922,-177.299,5.912,148.246
C07834=1235.190,202.565,-55.946,-177.297,5.914,148.246
C07835=1235.186,202.814,-55.970,-177.295,5.915,148.246
C07836=1235.181,203.062,-55.994,-177.292,5.917,148.245
C07837=1235.177,203.311,-56.018,-177.289,5.919,148.245
C07838=1235.171,203.560,-56.042,-177.287,5.921,148.245
C07839=1235.168,203.809,-56.066,-177.284,5.921,148.244
C07840=1235.163,204.058,-56.090,-177.282,5.923,148.244
C07841=1235.159,204.307,-56.114,-177.279,5.925,148.243
C07842=1235.154,204.555,-56.138,-177.277,5.926,148.243
C07843=1235.149,204.804,-56.162,-177.274,5.928,148.243
C07844=1235.144,205.053,-56.186,-177.272,5.930,148.242
C07845=1235.140,205.302,-56.210,-177.269,5.932,148.242
C07846=1235.136,205.551,-56.234,-177.266,5.932,148.241
C07847=1235.131,205.800,-56.258,-177.264,5.934,148.241
C07848=1235.126,206.048,-56.282,-177.261,5.936,148.241
C07849=1235.122,206.297,-56.306,-177.259,5.937,148.240
C07850=1235.117,206.545,-56.330,-177.257,5.939,148.240
C07851=1235.113,206.795,-56.355,-177.254,5.941,148.240
C07852=1235.108,207.043,-56.379,-177.251,5.943,148.239
C07853=1235.104,207.292,-56.402,-177.249,5.943,148.239
C07854=1235.099,207.541,-56.426,-177.246,5.945,148.238
C07855=1235.094,207.789,-56.451,-177.243,5.947,148.238
C07856=1235.090,208.039,-56.476,-177.241,5.949,148.238
C07857=1235.086,208.288,-56.499,-177.239,5.950,148.237
C07858=1235.080,208.536,-56.524,-177.236,5.952,148.237
C07859=1235.076,208.785,-56.548,-177.233,5.954,148.237
C07860=1235.072,209.033,-56.572,-177.231,5.955,148.236
C07861=1235.067,209.283,-56.597,-177.228,5.956,148.236
C07862=1235.063,209.531,-56.621,-177.226,5.958,148.235
C07863=1235.058,209.780,-56.644,-177.223,5.960,148.235
C07864=1235.053,210.029,-56.669,-177.221,5.961,148.235
C07865=1235.049,210.278,-56.693,-177.218,5.963,148.234
C07866=1235.044,210.527,-56.718,-177.216,5.965,148.234
C07867=1235.040,210.775,-56.742,-177.213,5.967,148.234
C07868=1235.035,211.023,-56.766,-177.211,5.968,148.233
C07869=1235.031,211.273,-56.791,-177.208,5.969,148.233
C07870=1235.025,211.544,-56.817,-177.205,5.971,148.232
C07871=1235.021,211.813,-56.843,-177.203,5.973,148.232
C07872=1235.016,212.084,-56.870,-177.200,5.975,148.232
C07873=1235.010,212.354,-56.897,-177.197,5.976,148.231
C07874=1235.007,212.603,-56.921,-177.194,5.978,148.231
C07875=1235.002,212.852,-56.946,-177.192,5.980,148.230
C07876=1234.997,213.100,-56.970,-177.189,5.982,148.230
C07877=1234.993,213.349,-56.995,-177.187,5.983,148.230
C07878=1234.988,213.598,-57.019,-177.184,5.985,148.229
C07879=1234.983,213.847,-57.044,-177.182,5.987,148.229
C07880=1234.979,214.096,-57.068,-177.179,5.989,148.229
C07881=1234.974,214.344,-57.093,-177.177,5.990,148.228
C07882=1234.970,214.593,-57.117,-177.174,5.991,148.228
C07883=1234.965,214.842,-57.142,-177.171,5.993,148.228
C07884=1234.961,215.091,-57.166,-177.169,5.995,148.227
C07885=1234.956,215.339,-57.191,-177.166,5.997,148.227
C07886=1234.952,215.589,-57.215,-177.164,5.998,148.227
C07887=1234.947,215.837,-57.240,-177.161,6.000,148.226
C07888=1234.942,216.086,-57.264,-177.159,6.002,148.226
C07889=1234.938,216.334,-57.290,-177.156,6.004,148.226
C07890=1234.934,216.583,-57.314,-177.153,6.005,148.225
C07891=1234.929,216.832,-57.338,-177.151,6.006,148.225
C07892=1234.925,217.081,-57.363,-177.149,6.008,148.225
C07893=1234.920,217.329,-57.387,-177.146,6.010,148.224
C07894=1234.915,217.578,-57.412,-177.143,6.012,148.224
C07895=1234.911,217.827,-57.437,-177.140,6.014,148.223
C07896=1234.906,218.075,-57.462,-177.138,6.015,148.223
C07897=1234.902,218.324,-57.486,-177.136,6.016,148.223
C07898=1234.897,218.573,-57.511,-177.133,6.018,148.222
C07899=1234.892,218.822,-57.536,-177.130,6.020,148.222
C07900=1234.888,219.070,-57.561,-177.128,6.022,148.222
C07901=1234.883,219.319,-57.586,-177.126,6.023,148.221
C07902=1234.879,219.568,-57.610,-177.123,6.025,148.221
C07903=1234.875,219.816,-57.635,-177.120,6.027,148.221
C07904=1234.870,220.065,-57.660,-177.118,6.029,148.220
C07905=1234.866,220.314,-57.684,-177.115,6.031,148.220
C07906=1234.861,220.563,-57.709,-177.113,6.032,148.220
C07907=1234.856,220.812,-57.735,-177.111,6.034,148.219
C07908=1234.852,221.060,-57.759,-177.108,6.035,148.219
C07909=1234.847,221.310,-57.784,-177.105,6.037,148.219
C07910=1234.843,221.558,-57.809,-177.103,6.039,148.218
C07911=1234.838,221.806,-57.833,-177.101,6.040,148.218
C07912=1234.834,222.055,-57.859,-177.097,6.042,148.217
C07913=1234.829,222.304,-57.884,-177.095,6.044,148.217
C07914=1234.825,222.553,-57.908,-177.092,6.046,148.217
C07915=1234.820,222.801,-57.934,-177.090,6.047,148.216
C07916=1234.816,223.050,-57.959,-177.088,6.048,148.216
C07917=1234.811,223.298,-57.984,-177.085,6.050,148.216
C07918=1234.807,223.547,-58.009,-177.082,6.052,148.215
C07919=1234.802,223.796,-58.033,-177.080,6.054,148.215
C07920=1234.798,224.045,-58.059,-177.077,6.056,148.215
C07921=1234.793,224.294,-58.084,-177.074,6.058,148.214
C07922=1234.789,224.542,-58.109,-177.072,6.059,148.214
C07923=1234.784,224.791,-58.133,-177.070,6.061,148.214
C07924=1234.780,225.040,-58.159,-177.067,6.063,148.213
C07925=1234.775,225.288,-58.184,-177.065,6.064,148.213
C07926=1234.770,225.537,-58.210,-177.062,6.066,148.213
C07927=1234.766,225.786,-58.234,-177.059,6.068,148.212
C07928=1234.762,226.034,-58.259,-177.057,6.069,148.212
C07929=1234.757,226.283,-58.284,-177.055,6.071,148.212
C07930=1234.752,226.532,-58.310,-177.052,6.073,148.211
C07931=1234.748,226.780,-58.335,-177.049,6.075,148.211
C07932=1234.743,227.030,-58.360,-177.047,6.077,148.211
C07933=1234.739,227.277,-58.385,-177.044,6.079,148.210
C07934=1234.734,227.527,-58.410,-177.042,6.080,148.210
C07935=1234.730,227.775,-58.436,-177.039,6.082,148.210
C07936=1234.725,228.024,-58.461,-177.037,6.083,148.209
C07937=1234.720,228.272,-58.486,-177.034,6.085,148.209
C07938=1234.716,228.521,-58.512,-177.032,6.087,148.209
C07939=1234.712,228.770,-58.537,-177.029,6.089,148.208
C07940=1234.707,229.019,-58.562,-177.027,6.090,148.208
C07941=1234.703,229.267,-58.587,-177.024,6.092,148.208
C07942=1234.698,229.515,-58.613,-177.022,6.094,148.207
C07943=1234.694,229.765,-58.638,-177.019,6.096,148.207
C07944=1234.690,230.014,-58.663,-177.016,6.098,148.207
C07945=1234.685,230.262,-58.689,-177.014,6.100,148.207
C07946=1234.681,230.510,-58.715,-177.012,6.101,148.206
C07947=1234.675,230.759,-58.739,-177.010,6.103,148.206
C07948=1234.671,231.008,-58.765,-177.007,6.105,148.206
C07949=1234.667,231.257,-58.791,-177.004,6.107,148.205
C07950=1234.662,231.505,-58.816,-177.002,6.108,148.205
C07951=1234.658,231.754,-58.841,-176.999,6.110,148.205
C07952=1234.653,232.002,-58.867,-176.997,6.112,148.204
C07953=1234.649,232.251,-58.892,-176.994,6.113,148.204
C07954=1234.644,232.500,-58.918,-176.992,6.115,148.204
C07955=1234.640,232.748,-58.943,-176.989,6.117,148.203
C07956=1234.635,232.998,-58.968,-176.987,6.119,148.203
C07957=1234.631,233.246,-58.994,-176.984,6.121,148.203
C07958=1234.626,233.494,-59.020,-176.981,6.123,148.203
C07959=1234.622,233.743,-59.045,-176.979,6.124,148.202
C07960=1234.617,233.992,-59.071,-176.977,6.126,148.202
C07961=1234.613,234.240,-59.096,-176.974,6.127,148.202
C07962=1234.608,234.489,-59.122,-176.971,6.129,148.201
C07963=1234.604,234.738,-59.148,-176.969,6.131,148.201
C07964=1234.599,234.986,-59.173,-176.966,6.133,148.201
C07965=1234.595,235.235,-59.198,-176.964,6.135,148.200
C07966=1234.591,235.484,-59.224,-176.961,6.137,148.200
C07967=1234.585,235.733,-59.250,-176.959,6.139,148.200
C07968=1234.581,235.981,-59.276,-176.957,6.140,148.199
C07969=1234.577,236.230,-59.302,-176.954,6.142,148.199
C07970=1234.572,236.478,-59.327,-176.952,6.144,148.199
C07971=1234.568,236.727,-59.353,-176.949,6.146,148.199
C07972=1234.563,236.976,-59.379,-176.946,6.148,148.198
C07973=1234.559,237.224,-59.404,-176.944,6.149,148.198
C07974=1234.554,237.495,-59.433,-176.941,6.151,148.198
C07975=1234.549,237.767,-59.461,-176.939,6.153,148.197
C07976=1234.544,238.038,-59.488,-176.936,6.155,148.197
C07977=1234.540,238.310,-59.517,-176.933,6.157,148.197
C07978=1234.534,238.558,-59.543,-176.931,6.159,148.196
C07979=1234.530,238.807,-59.569,-176.928,6.161,148.196
C07980=1234.526,239.056,-59.595,-176.925,6.163,148.196
C07981=1234.522,239.304,-59.620,-176.923,6.165,148.195
C07982=1234.517,239.553,-59.646,-176.920,6.166,148.195
C07983=1234.512,239.802,-59.672,-176.918,6.168,148.195
C07984=1234.508,240.050,-59.698,-176.915,6.170,148.194
C07985=1234.504,240.299,-59.724,-176.913,6.172,148.194
C07986=1234.499,240.547,-59.750,-176.911,6.173,148.194
C07987=1234.495,240.796,-59.775,-176.908,6.175,148.194
C07988=1234.490,241.045,-59.802,-176.906,6.177,148.193
C07989=1234.485,241.293,-59.828,-176.903,6.179,148.193
C07990=1234.481,241.542,-59.854,-176.900,6.181,148.193
C07991=1234.477,241.790,-59.879,-176.898,6.183,148.192
C07992=1234.472,242.039,-59.906,-176.895,6.185,148.192
C07993=1234.467,242.288,-59.931,-176.893,6.187,148.192
C07994=1234.463,242.537,-59.957,-176.890,6.189,148.192
C07995=1234.459,242.785,-59.984,-176.888,6.191,148.191
C07996=1234.454,243.033,-60.010,-176.885,6.193,148.191
C07997=1234.449,243.282,-60.035,-176.883,6.194,148.191
C07998=1234.446,243.530,-60.062,-176.881,6.196,148.190
C07999=1234.441,243.779,-60.088,-176.878,6.197,148.190
C08000=1234.436,244.028,-60.114,-176.876,6.200,148.190
C08001=1234.432,244.276,-60.140,-176.873,6.202,148.190
C08002=1234.427,244.525,-60.166,-176.871,6.203,148.189
C08003=1234.423,244.773,-60.192,-176.868,6.205,148.189
C08004=1234.418,245.022,-60.219,-176.865,6.207,148.189
C08005=1234.414,245.271,-60.245,-176.863,6.209,148.188
C08006=1234.410,245.520,-60.271,-176.860,6.211,148.188
C08007=1234.405,245.768,-60.298,-176.858,6.213,148.188
C08008=1234.401,246.017,-60.324,-176.855,6.215,148.188
C08009=1234.396,246.264,-60.350,-176.853,6.216,148.187
C08010=1234.391,246.513,-60.376,-176.851,6.218,148.187
C08011=1234.387,246.762,-60.402,-176.848,6.220,148.187
C08012=1234.382,247.011,-60.429,-176.846,6.222,148.187
C08013=1234.378,247.260,-60.455,-176.843,6.224,148.186
C08014=1234.374,247.508,-60.481,-176.841,6.226,148.186
C08015=1234.369,247.757,-60.507,-176.838,6.228,148.186
C08016=1234.365,248.005,-60.534,-176.836,6.230,148.185
C08017=1234.360,248.254,-60.560,-176.833,6.232,148.185
C08018=1234.356,248.502,-60.587,-176.830,6.233,148.185
C08019=1234.351,248.751,-60.613,-176.828,6.236,148.185
C08020=1234.347,248.999,-60.639,-176.826,6.238,148.184
C08021=1234.342,249.248,-60.665,-176.823,6.239,148.184
C08022=1234.338,249.496,-60.692,-176.820,6.241,148.184
C08023=1234.333,249.745,-60.718,-176.818,6.243,148.184
C08024=1234.329,249.994,-60.745,-176.816,6.245,148.183
C08025=1234.325,250.242,-60.772,-176.813,6.247,148.183
C08026=1234.320,250.491,-60.798,-176.811,6.248,148.183
C08027=1234.316,250.739,-60.825,-176.808,6.250,148.183
C08028=1234.311,250.988,-60.850,-176.806,6.252,148.182
C08029=1234.307,251.237,-60.877,-176.804,6.254,148.182
C08030=1234.303,251.485,-60.904,-176.801,6.256,148.182
C08031=1234.298,251.734,-60.930,-176.798,6.258,148.182
C08032=1234.294,251.982,-60.957,-176.796,6.260,148.181
C08033=1234.289,252.231,-60.984,-176.793,6.262,148.181
C08034=1234.284,252.480,-61.010,-176.791,6.264,148.181
C08035=1234.280,252.728,-61.037,-176.789,6.266,148.181
C08036=1234.276,252.976,-61.064,-176.786,6.268,148.180
C08037=1234.272,253.225,-61.089,-176.783,6.270,148.180
C08038=1234.267,253.474,-61.116,-176.781,6.272,148.180
C08039=1234.263,253.722,-61.143,-176.779,6.274,148.180
C08040=1234.258,253.970,-61.170,-176.776,6.276,148.179
C08041=1234.253,254.219,-61.196,-176.773,6.278,148.179
C08042=1234.249,254.468,-61.223,-176.771,6.280,148.179
C08043=1234.245,254.716,-61.250,-176.769,6.282,148.179
C08044=1234.240,254.965,-61.277,-176.766,6.284,148.178
C08045=1234.236,255.213,-61.303,-176.763,6.286,148.178
C08046=1234.231,255.462,-61.330,-176.761,6.288,148.178
C08047=1234.227,255.710,-61.357,-176.759,6.290,148.178
C08048=1234.223,255.959,-61.383,-176.756,6.292,148.177
C08049=1234.218,256.207,-61.410,-176.754,6.294,148.177
C08050=1234.213,256.456,-61.437,-176.751,6.295,148.177
C08051=1234.209,256.704,-61.464,-176.749,6.298,148.177
C08052=1234.205,256.952,-61.491,-176.746,6.300,148.176
C08053=1234.200,257.201,-61.517,-176.744,6.301,148.176
C08054=1234.196,257.450,-61.544,-176.741,6.303,148.176
C08055=1234.191,257.698,-61.571,-176.739,6.306,148.176
C08056=1234.187,257.947,-61.598,-176.736,6.307,148.175
C08057=1234.182,258.195,-61.625,-176.734,6.309,148.175
C08058=1234.179,258.444,-61.652,-176.732,6.312,148.175
C08059=1234.174,258.692,-61.679,-176.729,6.313,148.175
C08060=1234.169,258.941,-61.706,-176.726,6.315,148.174
C08061=1234.165,259.189,-61.733,-176.724,6.317,148.174
C08062=1234.161,259.438,-61.759,-176.722,6.319,148.174
C08063=1234.156,259.686,-61.786,-176.719,6.321,148.174
C08064=1234.151,259.935,-61.814,-176.716,6.323,148.173
C08065=1234.147,260.183,-61.841,-176.714,6.325,148.173
C08066=1234.142,260.432,-61.868,-176.712,6.327,148.173
C08067=1234.138,260.680,-61.894,-176.709,6.329,148.173
C08068=1234.134,260.929,-61.922,-176.706,6.331,148.172
C08069=1234.129,261.178,-61.949,-176.704,6.333,148.172
C08070=1234.125,261.426,-61.976,-176.702,6.335,148.172
C08071=1234.120,261.675,-62.003,-176.699,6.337,148.172
C08072=1234.115,261.923,-62.030,-176.697,6.339,148.172
C08073=1234.112,262.171,-62.056,-176.694,6.341,148.171
C08074=1234.107,262.419,-62.084,-176.692,6.343,148.171
C08075=1234.103,262.668,-62.111,-176.690,6.345,148.171
C08076=1234.098,262.917,-62.139,-176.687,6.347,148.171
C08077=1234.094,263.165,-62.166,-176.685,6.349,148.170
C08078=1234.089,263.438,-62.195,-176.682,6.351,148.170
C08079=1234.084,263.710,-62.226,-176.680,6.353,148.170
C08080=1234.079,263.983,-62.255,-176.677,6.356,148.170
C08081=1234.075,264.255,-62.284,-176.674,6.358,148.169
C08082=1234.070,264.504,-62.311,-176.671,6.360,148.169
C08083=1234.066,264.752,-62.340,-176.669,6.362,148.169
C08084=1234.062,265.001,-62.367,-176.667,6.364,148.169
C08085=1234.057,265.249,-62.394,-176.664,6.366,148.168
C08086=1234.052,265.498,-62.421,-176.662,6.368,148.168
C08087=1234.048,265.746,-62.448,-176.659,6.370,148.168
C08088=1234.044,265.995,-62.476,-176.657,6.372,148.168
C08089=1234.039,266.244,-62.503,-176.655,6.374,148.168
C08090=1234.035,266.491,-62.531,-176.652,6.376,148.167
C08091=1234.030,266.740,-62.558,-176.650,6.378,148.167
C08092=1234.026,266.989,-62.585,-176.647,6.381,148.167
C08093=1234.022,267.237,-62.613,-176.644,6.383,148.167
C08094=1234.017,267.485,-62.640,-176.642,6.385,148.166
C08095=1234.013,267.734,-62.667,-176.640,6.387,148.166
C08096=1234.009,267.983,-62.695,-176.637,6.389,148.166
C08097=1234.004,268.231,-62.722,-176.635,6.391,148.166
C08098=1233.999,268.480,-62.749,-176.632,6.393,148.166
C08099=1233.995,268.727,-62.777,-176.630,6.395,148.165
C08100=1233.991,268.977,-62.805,-176.628,6.397,148.165
C08101=1233.987,269.224,-62.832,-176.625,6.399,148.165
C08102=1233.982,269.473,-62.859,-176.622,6.401,148.165
C08103=1233.977,269.721,-62.887,-176.620,6.403,148.165
C08104=1233.974,269.970,-62.915,-176.618,6.405,148.164
C08105=1233.968,270.219,-62.942,-176.616,6.407,148.164
C08106=1233.964,270.467,-62.970,-176.613,6.409,148.164
C08107=1233.960,270.716,-62.998,-176.610,6.411,148.164
C08108=1233.955,270.964,-63.025,-176.608,6.413,148.164
C08109=1233.951,271.212,-63.052,-176.605,6.416,148.163
C08110=1233.947,271.461,-63.080,-176.603,6.418,148.163
C08111=1233.942,271.709,-63.108,-176.600,6.420,148.163
C08112=1233.938,271.957,-63.135,-176.598,6.422,148.163
C08113=1233.933,272.207,-63.163,-176.596,6.424,148.163
C08114=1233.929,272.455,-63.191,-176.593,6.426,148.162
C08115=1233.925,272.703,-63.219,-176.591,6.428,148.162
C08116=1233.921,272.952,-63.246,-176.588,6.430,148.162
C08117=1233.916,273.200,-63.274,-176.586,6.432,148.162
C08118=1233.912,273.448,-63.301,-176.584,6.434,148.162
C08119=1233.907,273.697,-63.330,-176.581,6.436,148.161
C08120=1233.903,273.945,-63.358,-176.579,6.438,148.161
C08121=1233.898,274.193,-63.385,-176.576,6.440,148.161
C08122=1233.894,274.442,-63.413,-176.574,6.443,148.161
C08123=1233.890,274.690,-63.441,-176.571,6.445,148.161
C08124=1233.885,274.939,-63.468,-176.569,6.447,148.161
C08125=1233.881,275.187,-63.496,-176.566,6.449,148.160
C08126=1233.876,275.435,-63.524,-176.564,6.452,148.160
C08127=1233.872,275.684,-63.552,-176.562,6.453,148.160
C08128=1233.867,275.932,-63.580,-176.560,6.456,148.160
C08129=1233.863,276.180,-63.608,-176.557,6.458,148.160
C08130=1233.859,276.429,-63.636,-176.554,6.460,148.159
C08131=1233.855,276.677,-63.663,-176.552,6.462,148.159
C08132=1233.850,276.926,-63.692,-176.550,6.464,148.159
C08133=1233.846,277.174,-63.720,-176.547,6.467,148.159
C08134=1233.841,277.422,-63.747,-176.544,6.469,148.159
C08135=1233.837,277.671,-63.775,-176.542,6.471,148.159
C08136=1233.832,277.919,-63.803,-176.540,6.473,148.158
C08137=1233.828,278.168,-63.831,-176.538,6.475,148.158
C08138=1233.824,278.416,-63.859,-176.535,6.477,148.158
C08139=1233.820,278.665,-63.888,-176.533,6.479,148.158
C08140=1233.815,278.913,-63.916,-176.530,6.481,148.158
C08141=1233.811,279.162,-63.943,-176.528,6.483,148.157
C08142=1233.806,279.410,-63.971,-176.525,6.486,148.157
C08143=1233.802,279.658,-63.999,-176.523,6.488,148.157
C08144=1233.797,279.907,-64.028,-176.520,6.490,148.157
C08145=1233.793,280.155,-64.056,-176.518,6.492,148.157
C08146=1233.789,280.403,-64.084,-176.516,6.494,148.156
C08147=1233.784,280.651,-64.112,-176.514,6.496,148.156
C08148=1233.780,280.900,-64.140,-176.511,6.499,148.156
C08149=1233.776,281.148,-64.168,-176.509,6.501,148.156
C08150=1233.771,281.397,-64.197,-176.507,6.503,148.156
C08151=1233.767,281.645,-64.225,-176.504,6.505,148.156
C08152=1233.763,281.894,-64.253,-176.502,6.508,148.156
C08153=1233.758,282.141,-64.281,-176.499,6.510,148.155
C08154=1233.754,282.390,-64.310,-176.497,6.512,148.155
C08155=1233.749,282.638,-64.338,-176.494,6.514,148.155
C08156=1233.746,282.887,-64.366,-176.492,6.516,148.155
C08157=1233.741,283.135,-64.394,-176.490,6.518,148.155
C08158=1233.737,283.383,-64.422,-176.487,6.521,148.155
C08159=1233.732,283.632,-64.451,-176.485,6.523,148.155
C08160=1233.728,283.880,-64.479,-176.482,6.525,148.154
C08161=1233.724,284.129,-64.508,-176.480,6.527,148.154
C08162=1233.719,284.377,-64.535,-176.477,6.529,148.154
C08163=1233.715,284.626,-64.564,-176.475,6.531,148.154
C08164=1233.710,284.874,-64.592,-176.473,6.533,148.154
C08165=1233.706,285.122,-64.621,-176.471,6.536,148.154
C08166=1233.702,285.370,-64.649,-176.468,6.539,148.154
C08167=1233.697,285.619,-64.678,-176.465,6.540,148.153
C08168=1233.692,285.867,-64.706,-176.463,6.543,148.153
C08169=1233.689,286.116,-64.734,-176.461,6.545,148.153
C08170=1233.684,286.364,-64.763,-176.459,6.547,148.153
C08171=1233.680,286.612,-64.792,-176.457,6.549,148.153
C08172=1233.675,286.861,-64.820,-176.453,6.552,148.153
C08173=1233.671,287.108,-64.848,-176.451,6.554,148.152
C08174=1233.667,287.357,-64.877,-176.449,6.556,148.152
C08175=1233.662,287.606,-64.905,-176.447,6.558,148.152
C08176=1233.658,287.853,-64.934,-176.444,6.560,148.152
C08177=1233.654,288.102,-64.963,-176.442,6.562,148.152
C08178=1233.649,288.350,-64.991,-176.440,6.565,148.152
C08179=1233.645,288.599,-65.020,-176.437,6.568,148.152
C08180=1233.641,288.847,-65.049,-176.435,6.569,148.151
C08181=1233.636,289.095,-65.076,-176.432,6.572,148.151
C08182=1233.631,289.370,-65.108,-176.430,6.574,148.151
C08183=1233.627,289.643,-65.140,-176.427,6.577,148.151
C08184=1233.622,289.917,-65.172,-176.425,6.579,148.151
C08185=1233.617,290.191,-65.203,-176.422,6.582,148.151
C08186=1233.613,290.440,-65.232,-176.420,6.584,148.151
C08187=1233.609,290.688,-65.261,-176.417,6.586,148.150
C08188=1233.604,290.936,-65.289,-176.415,6.588,148.150
C08189=1233.599,291.185,-65.318,-176.413,6.591,148.150
C08190=1233.595,291.433,-65.347,-176.410,6.593,148.150
C08191=1233.591,291.681,-65.375,-176.408,6.595,148.150
C08192=1233.587,291.930,-65.405,-176.406,6.597,148.150
C08193=1233.583,292.178,-65.433,-176.403,6.599,148.150
C08194=1233.578,292.426,-65.462,-176.401,6.602,148.150
C08195=1233.574,292.675,-65.491,-176.398,6.605,148.150
C08196=1233.569,292.923,-65.520,-176.396,6.607,148.149
C08197=1233.565,293.171,-65.548,-176.394,6.609,148.149
C08198=1233.561,293.419,-65.577,-176.392,6.611,148.149
C08199=1233.556,293.668,-65.606,-176.389,6.613,148.149
C08200=1233.552,293.916,-65.635,-176.386,6.616,148.149
C08201=1233.547,294.165,-65.664,-176.384,6.618,148.149
C08202=1233.544,294.412,-65.693,-176.382,6.620,148.149
C08203=1233.539,294.661,-65.722,-176.380,6.622,148.149
C08204=1233.534,294.909,-65.751,-176.377,6.625,148.148
C08205=1233.530,295.158,-65.779,-176.375,6.627,148.148
C08206=1233.526,295.406,-65.809,-176.373,6.630,148.148
C08207=1233.522,295.654,-65.838,-176.370,6.632,148.148
C08208=1233.517,295.902,-65.866,-176.368,6.634,148.148
C08209=1233.513,296.150,-65.896,-176.366,6.636,148.148
C08210=1233.509,296.399,-65.925,-176.364,6.638,148.148
C08211=1233.504,296.648,-65.954,-176.361,6.641,148.148
C08212=1233.499,296.895,-65.983,-176.359,6.643,148.148
C08213=1233.496,297.143,-66.012,-176.356,6.646,148.148
C08214=1233.492,297.392,-66.040,-176.354,6.648,148.148
C08215=1233.487,297.640,-66.070,-176.352,6.650,148.147
C08216=1233.483,297.888,-66.099,-176.349,6.653,148.147
C08217=1233.478,298.137,-66.128,-176.347,6.655,148.147
C08218=1233.474,298.385,-66.157,-176.345,6.657,148.147
C08219=1233.470,298.633,-66.187,-176.343,6.659,148.147
C08220=1233.466,298.882,-66.216,-176.340,6.661,148.147
C08221=1233.460,299.130,-66.244,-176.338,6.664,148.147
C08222=1233.456,299.378,-66.274,-176.335,6.667,148.147
C08223=1233.452,299.626,-66.303,-176.333,6.669,148.147
C08224=1233.448,299.875,-66.333,-176.331,6.671,148.147
C08225=1233.444,300.123,-66.362,-176.329,6.673,148.146
C08226=1233.440,300.371,-66.390,-176.326,6.676,148.146
C08227=1233.435,300.619,-66.420,-176.324,6.678,148.146
C08228=1233.431,300.867,-66.449,-176.322,6.681,148.146
C08229=1233.427,301.115,-66.478,-176.320,6.683,148.146
C08230=1233.423,301.364,-66.508,-176.318,6.685,148.146
C08231=1233.418,301.612,-66.537,-176.314,6.688,148.146
C08232=1233.414,301.861,-66.566,-176.312,6.690,148.146
C08233=1233.409,302.108,-66.595,-176.310,6.692,148.146
C08234=1233.404,302.357,-66.625,-176.308,6.694,148.146
C08235=1233.400,302.605,-66.655,-176.306,6.697,148.146
C08236=1233.396,302.854,-66.684,-176.303,6.700,148.146
C08237=1233.392,303.102,-66.714,-176.301,6.702,148.146
C08238=1233.388,303.350,-66.743,-176.299,6.704,148.146
C08239=1233.383,303.598,-66.772,-176.297,6.706,148.145
C08240=1233.379,303.847,-66.802,-176.294,6.709,148.145
C08241=1233.374,304.094,-66.831,-176.292,6.711,148.145
C08242=1233.370,304.343,-66.860,-176.290,6.714,148.145
C08243=1233.366,304.591,-66.890,-176.288,6.716,148.145
C08244=1233.362,304.839,-66.919,-176.286,6.718,148.145
C08245=1233.358,305.087,-66.949,-176.283,6.721,148.145
C08246=1233.354,305.336,-66.978,-176.281,6.723,148.145
C08247=1233.349,305.584,-67.008,-176.279,6.726,148.145
C08248=1233.344,305.832,-67.038,-176.277,6.728,148.145
C08249=1233.340,306.081,-67.067,-176.274,6.731,148.145
C08250=1233.336,306.329,-67.097,-176.271,6.733,148.145
C08251=1233.331,306.577,-67.126,-176.269,6.735,148.145
C08252=1233.327,306.825,-67.155,-176.267,6.737,148.145
C08253=1233.323,307.072,-67.185,-176.265,6.739,148.145
C08254=1233.318,307.321,-67.215,-176.262,6.743,148.145
C08255=1233.314,307.569,-67.245,-176.260,6.745,148.144
C08256=1233.310,307.818,-67.274,-176.258,6.747,148.144
C08257=1233.306,308.066,-67.304,-176.256,6.749,148.144
C08258=1233.302,308.314,-67.333,-176.254,6.752,148.144
C08259=1233.297,308.562,-67.364,-176.251,6.754,148.144
C08260=1233.293,308.810,-67.393,-176.249,6.757,148.144
C08261=1233.289,309.059,-67.423,-176.247,6.759,148.144
C08262=1233.284,309.307,-67.452,-176.245,6.762,148.144
C08263=1233.279,309.555,-67.482,-176.242,6.764,148.144
C08264=1233.276,309.803,-67.513,-176.240,6.766,148.144
C08265=1233.271,310.051,-67.542,-176.238,6.769,148.144
C08266=1233.267,310.300,-67.571,-176.236,6.771,148.144
C08267=1233.262,310.548,-67.602,-176.234,6.774,148.144
C08268=1233.258,310.796,-67.632,-176.231,6.776,148.144
C08269=1233.254,311.044,-67.661,-176.229,6.778,148.144
C08270=1233.250,311.292,-67.691,-176.227,6.781,148.144
C08271=1233.245,311.540,-67.721,-176.225,6.784,148.144
C08272=1233.241,311.789,-67.751,-176.222,6.786,148.144
C08273=1233.237,312.037,-67.780,-176.220,6.788,148.144
C08274=1233.233,312.285,-67.811,-176.218,6.790,148.144
C08275=1233.228,312.533,-67.841,-176.216,6.793,148.144
C08276=1233.224,312.781,-67.870,-176.214,6.796,148.144
C08277=1233.220,313.029,-67.901,-176.211,6.798,148.144
C08278=1233.215,313.278,-67.930,-176.209,6.800,148.144
C08279=1233.211,313.525,-67.960,-176.207,6.803,148.144
C08280=1233.207,313.774,-67.990,-176.205,6.805,148.144
C08281=1233.202,314.022,-68.020,-176.203,6.808,148.144
C08282=1233.199,314.270,-68.050,-176.201,6.810,148.144
C08283=1233.194,314.519,-68.080,-176.198,6.813,148.144
C08284=1233.190,314.767,-68.111,-176.196,6.815,148.144
C08285=1233.185,315.015,-68.141,-176.194,6.818,148.144
C08286=1233.181,315.290,-68.174,-176.191,6.821,148.144
C08287=1233.176,315.566,-68.207,-176.189,6.823,148.143
C08288=1233.172,315.842,-68.241,-176.187,6.826,148.143
C08289=1233.167,316.117,-68.274,-176.185,6.828,148.143
C08290=1233.162,316.365,-68.305,-176.182,6.831,148.143
C08291=1233.158,316.613,-68.334,-176.180,6.834,148.143
C08292=1233.154,316.862,-68.365,-176.178,6.836,148.143
C08293=1233.150,317.110,-68.395,-176.176,6.838,148.143
C08294=1233.145,317.358,-68.425,-176.173,6.841,148.144
C08295=1233.141,317.606,-68.456,-176.171,6.844,148.143
C08296=1233.136,317.855,-68.486,-176.169,6.846,148.143
C08297=1233.132,318.102,-68.516,-176.167,6.848,148.143
C08298=1233.127,318.351,-68.546,-176.165,6.851,148.143
C08299=1233.124,318.598,-68.576,-176.162,6.853,148.143
C08300=1233.120,318.847,-68.607,-176.161,6.856,148.144
C08301=1233.115,319.095,-68.637,-176.159,6.858,148.143
C08302=1233.111,319.343,-68.667,-176.156,6.861,148.143
C08303=1233.107,319.591,-68.697,-176.154,6.863,148.143
C08304=1233.102,319.840,-68.728,-176.152,6.866,148.143
C08305=1233.098,320.087,-68.758,-176.150,6.868,148.144
C08306=1233.094,320.336,-68.789,-176.148,6.871,148.144
C08307=1233.090,320.584,-68.818,-176.146,6.874,148.144
C08308=1233.085,320.832,-68.849,-176.143,6.876,148.143
C08309=1233.081,321.080,-68.879,-176.141,6.878,148.143
C08310=1233.077,321.328,-68.910,-176.139,6.881,148.144
C08311=1233.072,321.576,-68.940,-176.137,6.884,148.144
C08312=1233.069,321.825,-68.971,-176.135,6.886,148.144
C08313=1233.064,322.073,-69.001,-176.133,6.888,148.144
C08314=1233.060,322.320,-69.032,-176.131,6.891,148.144
C08315=1233.056,322.568,-69.062,-176.129,6.894,148.144
C08316=1233.051,322.817,-69.093,-176.127,6.896,148.144
C08317=1233.047,323.065,-69.123,-176.125,6.898,148.144
C08318=1233.043,323.313,-69.154,-176.122,6.901,148.144
C08319=1233.039,323.561,-69.184,-176.120,6.904,148.144
C08320=1233.034,323.809,-69.215,-176.118,6.906,148.144
C08321=1233.030,324.057,-69.246,-176.116,6.908,148.144
C08322=1233.026,324.305,-69.276,-176.114,6.912,148.144
C08323=1233.022,324.553,-69.307,-176.112,6.914,148.144
C08324=1233.017,324.802,-69.337,-176.110,6.916,148.144
C08325=1233.014,325.050,-69.367,-176.108,6.919,148.144
C08326=1233.009,325.298,-69.398,-176.105,6.922,148.144
C08327=1233.004,325.546,-69.429,-176.104,6.924,148.144
C08328=1233.000,325.793,-69.459,-176.102,6.926,148.144
C08329=1232.996,326.042,-69.490,-176.100,6.929,148.144
C08330=1232.992,326.290,-69.521,-176.097,6.932,148.144
C08331=1232.987,326.538,-69.552,-176.095,6.934,148.144
C08332=1232.984,326.786,-69.582,-176.093,6.936,148.144
C08333=1232.979,327.034,-69.613,-176.092,6.939,148.144
C08334=1232.975,327.282,-69.644,-176.089,6.942,148.144
C08335=1232.970,327.530,-69.674,-176.087,6.944,148.144
C08336=1232.967,327.779,-69.705,-176.085,6.947,148.145
C08337=1232.962,328.027,-69.736,-176.083,6.949,148.145
C08338=1232.958,328.275,-69.766,-176.081,6.952,148.145
C08339=1232.954,328.523,-69.798,-176.079,6.955,148.145
C08340=1232.950,328.771,-69.828,-176.077,6.957,148.145
C08341=1232.945,329.018,-69.859,-176.075,6.959,148.145
C08342=1232.941,329.267,-69.890,-176.072,6.962,148.145
C08343=1232.937,329.515,-69.921,-176.071,6.965,148.145
C08344=1232.932,329.763,-69.952,-176.069,6.967,148.145
C08345=1232.929,330.011,-69.982,-176.067,6.969,148.145
C08346=1232.924,330.259,-70.013,-176.065,6.972,148.145
C08347=1232.920,330.507,-70.044,-176.062,6.975,148.145
C08348=1232.916,330.756,-70.075,-176.061,6.978,148.145
C08349=1232.911,331.003,-70.107,-176.059,6.980,148.145
C08350=1232.907,331.251,-70.137,-176.057,6.982,148.145
C08351=1232.903,331.500,-70.168,-176.054,6.985,148.146
C08352=1232.899,331.747,-70.199,-176.053,6.988,148.146
C08353=1232.894,331.995,-70.229,-176.051,6.990,148.146
C08354=1232.891,332.243,-70.261,-176.049,6.993,148.146
C08355=1232.886,332.491,-70.292,-176.046,6.996,148.146
C08356=1232.881,332.739,-70.323,-176.045,6.998,148.146
C08357=1232.877,332.988,-70.354,-176.043,7.001,148.146
C08358=1232.873,333.235,-70.385,-176.041,7.003,148.146
C08359=1232.869,333.484,-70.416,-176.038,7.006,148.146
C08360=1232.864,333.732,-70.447,-176.037,7.009,148.146
C08361=1232.860,333.979,-70.479,-176.035,7.011,148.146
C08362=1232.857,334.227,-70.509,-176.033,7.013,148.146
C08363=1232.852,334.475,-70.540,-176.031,7.017,148.146
C08364=1232.848,334.723,-70.572,-176.029,7.019,148.147
C08365=1232.844,334.971,-70.603,-176.027,7.021,148.147
C08366=1232.839,335.219,-70.633,-176.025,7.024,148.147
C08367=1232.836,335.467,-70.665,-176.024,7.026,148.147
C08368=1232.831,335.715,-70.696,-176.021,7.029,148.147
C08369=1232.827,335.963,-70.728,-176.019,7.032,148.147
C08370=1232.823,336.211,-70.759,-176.017,7.034,148.147
C08371=1232.819,336.460,-70.790,-176.016,7.037,148.147
C08372=1232.814,336.707,-70.821,-176.013,7.040,148.147
C08373=1232.810,336.956,-70.852,-176.011,7.042,148.148
C08374=1232.806,337.203,-70.884,-176.010,7.045,148.148
C08375=1232.801,337.451,-70.915,-176.008,7.047,148.148
C08376=1232.798,337.699,-70.946,-176.005,7.050,148.148
C08377=1232.793,337.947,-70.977,-176.004,7.053,148.148
C08378=1232.789,338.195,-71.009,-176.002,7.055,148.148
C08379=1232.785,338.443,-71.040,-176.000,7.058,148.148
C08380=1232.780,338.692,-71.072,-175.998,7.060,148.148
C08381=1232.776,338.940,-71.103,-175.996,7.063,148.148
C08382=1232.772,339.188,-71.135,-175.994,7.066,148.149
C08383=1232.767,339.436,-71.166,-175.993,7.068,148.149
C08384=1232.764,339.684,-71.197,-175.991,7.071,148.149
C08385=1232.759,339.932,-71.228,-175.989,7.073,148.149
C08386=1232.755,340.180,-71.260,-175.987,7.077,148.149
C08387=1232.751,340.428,-71.291,-175.985,7.079,148.149
C08388=1232.747,340.676,-71.323,-175.983,7.081,148.149
C08389=1232.743,340.923,-71.354,-175.981,7.084,148.149
C08390=1232.738,341.201,-71.389,-175.979,7.087,148.150
C08391=1232.733,341.478,-71.424,-175.977,7.090,148.150
C08392=1232.728,341.756,-71.460,-175.975,7.093,148.150
C08393=1232.723,342.034,-71.495,-175.972,7.096,148.150
C08394=1232.719,342.281,-71.527,-175.971,7.098,148.150
C08395=1232.715,342.530,-71.558,-175.969,7.101,148.150
C08396=1232.711,342.777,-71.589,-175.967,7.104,148.150
C08397=1232.707,343.025,-71.621,-175.965,7.107,148.151
C08398=1232.702,343.273,-71.653,-175.963,7.109,148.151
C08399=1232.698,343.522,-71.685,-175.962,7.112,148.151
C08400=1232.694,343.769,-71.716,-175.960,7.114,148.151
C08401=1232.690,344.017,-71.748,-175.958,7.117,148.151
C08402=1232.686,344.266,-71.779,-175.956,7.120,148.151
C08403=1232.681,344.513,-71.811,-175.954,7.122,148.151
C08404=1232.677,344.761,-71.843,-175.952,7.125,148.152
C08405=1232.673,345.009,-71.874,-175.951,7.127,148.152
C08406=1232.669,345.257,-71.906,-175.949,7.130,148.152
C08407=1232.664,345.505,-71.938,-175.947,7.133,148.152
C08408=1232.660,345.753,-71.969,-175.945,7.136,148.152
C08409=1232.656,346.001,-72.001,-175.943,7.138,148.152
C08410=1232.652,346.248,-72.033,-175.942,7.141,148.153
C08411=1232.648,346.497,-72.065,-175.940,7.143,148.153
C08412=1232.643,346.745,-72.096,-175.938,7.146,148.153
C08413=1232.639,346.993,-72.128,-175.936,7.149,148.153
C08414=1232.635,347.241,-72.160,-175.935,7.152,148.153
C08415=1232.631,347.488,-72.192,-175.933,7.154,148.154
C08416=1232.627,347.736,-72.224,-175.931,7.156,148.153
C08417=1232.623,347.984,-72.255,-175.929,7.159,148.154
C08418=1232.618,348.232,-72.288,-175.927,7.162,148.154
C08419=1232.615,348.480,-72.319,-175.926,7.165,148.154
C08420=1232.610,348.728,-72.351,-175.924,7.167,148.154
C08421=1232.606,348.976,-72.383,-175.922,7.170,148.154
C08422=1232.602,349.225,-72.414,-175.921,7.172,148.155
C08423=1232.597,349.472,-72.446,-175.919,7.175,148.155
C08424=1232.593,349.720,-72.478,-175.917,7.178,148.155
C08425=1232.589,349.968,-72.510,-175.915,7.181,148.155
C08426=1232.584,350.216,-72.542,-175.914,7.183,148.155
C08427=1232.581,350.464,-72.574,-175.912,7.186,148.156
C08428=1232.577,350.712,-72.606,-175.910,7.188,148.156
C08429=1232.572,350.960,-72.638,-175.909,7.191,148.156
C08430=1232.568,351.208,-72.670,-175.907,7.193,148.156
C08431=1232.564,351.456,-72.702,-175.905,7.197,148.156
C08432=1232.560,351.703,-72.734,-175.903,7.199,148.157
C08433=1232.556,351.951,-72.766,-175.902,7.202,148.157
C08434=1232.551,352.199,-72.799,-175.900,7.204,148.157
C08435=1232.547,352.446,-72.830,-175.899,7.207,148.157
C08436=1232.543,352.695,-72.863,-175.897,7.209,148.157
C08437=1232.539,352.943,-72.895,-175.895,7.212,148.157
C08438=1232.534,353.191,-72.927,-175.893,7.215,148.158
C08439=1232.530,353.439,-72.958,-175.892,7.218,148.158
C08440=1232.527,353.687,-72.990,-175.890,7.220,148.158
C08441=1232.522,353.934,-73.022,-175.888,7.223,148.158
C08442=1232.518,354.182,-73.055,-175.887,7.226,148.158
C08443=1232.514,354.430,-73.087,-175.885,7.228,148.159
C08444=1232.510,354.678,-73.119,-175.883,7.231,148.159
C08445=1232.505,354.926,-73.151,-175.882,7.234,148.159
C08446=1232.501,355.174,-73.183,-175.880,7.237,148.159
C08447=1232.497,355.422,-73.216,-175.878,7.239,148.160
C08448=1232.493,355.670,-73.248,-175.877,7.242,148.160
C08449=1232.488,355.917,-73.280,-175.875,7.244,148.160
C08450=1232.485,356.165,-73.312,-175.874,7.247,148.160
C08451=1232.480,356.414,-73.344,-175.872,7.249,148.160
C08452=1232.477,356.661,-73.377,-175.871,7.252,148.161
C08453=1232.472,356.909,-73.409,-175.869,7.255,148.161
C08454=1232.467,357.157,-73.442,-175.867,7.258,148.161
C08455=1232.464,357.405,-73.473,-175.865,7.261,148.161
C08456=1232.459,357.653,-73.507,-175.864,7.263,148.162
C08457=1232.455,357.900,-73.538,-175.862,7.266,148.162
C08458=1232.451,358.148,-73.570,-175.861,7.269,148.162
C08459=1232.447,358.396,-73.603,-175.859,7.271,148.162
C08460=1232.443,358.644,-73.635,-175.858,7.274,148.163
C08461=1232.438,358.893,-73.668,-175.856,7.276,148.163
C08462=1232.434,359.139,-73.700,-175.855,7.279,148.163
C08463=1232.430,359.388,-73.733,-175.853,7.282,148.163
C08464=1232.426,359.636,-73.764,-175.851,7.285,148.164
C08465=1232.422,359.883,-73.798,-175.850,7.287,148.164
C08466=1232.418,360.132,-73.830,-175.848,7.290,148.164
C08467=1232.414,360.378,-73.862,-175.847,7.293,148.164
C08468=1232.409,360.627,-73.895,-175.845,7.295,148.165
C08469=1232.406,360.875,-73.926,-175.844,7.298,148.165
C08470=1232.401,361.123,-73.960,-175.842,7.301,148.165
C08471=1232.397,361.371,-73.992,-175.841,7.303,148.165
C08472=1232.393,361.618,-74.024,-175.839,7.306,148.165
C08473=1232.388,361.866,-74.057,-175.838,7.309,148.166
C08474=1232.384,362.114,-74.090,-175.836,7.311,148.166
C08475=1232.381,362.362,-74.122,-175.835,7.314,148.166
C08476=1232.377,362.609,-74.155,-175.834,7.317,148.167
C08477=1232.372,362.858,-74.187,-175.832,7.319,148.167
C08478=1232.367,363.105,-74.220,-175.830,7.322,148.167
C08479=1232.364,363.353,-74.252,-175.829,7.324,148.167
C08480=1232.359,363.601,-74.285,-175.827,7.328,148.168
C08481=1232.355,363.849,-74.318,-175.825,7.330,148.168
C08482=1232.352,364.096,-74.350,-175.824,7.333,148.168
C08483=1232.347,364.345,-74.383,-175.823,7.336,148.168
C08484=1232.343,364.592,-74.416,-175.821,7.339,148.169
C08485=1232.339,364.841,-74.448,-175.820,7.341,148.169
C08486=1232.335,365.088,-74.480,-175.818,7.344,148.169
C08487=1232.330,365.336,-74.513,-175.817,7.346,148.170
C08488=1232.326,365.584,-74.546,-175.815,7.349,148.170
C08489=1232.323,365.831,-74.579,-175.814,7.352,148.170
C08490=1232.318,366.079,-74.611,-175.813,7.354,148.170
C08491=1232.314,366.327,-74.644,-175.812,7.357,148.171
C08492=1232.310,366.575,-74.677,-175.810,7.360,148.171
C08493=1232.305,366.823,-74.710,-175.809,7.362,148.171
C08494=1232.301,367.102,-74.746,-175.807,7.365,148.172
C08495=1232.296,367.382,-74.783,-175.806,7.368,148.172
C08496=1232.291,367.662,-74.821,-175.804,7.371,148.172
C08497=1232.287,367.940,-74.857,-175.803,7.374,148.173
C08498=1232.283,368.188,-74.890,-175.801,7.377,148.173
C08499=1232.278,368.436,-74.923,-175.800,7.379,148.173
C08500=1232.274,368.684,-74.956,-175.798,7.382,148.173
C08501=1232.271,368.931,-74.988,-175.797,7.385,148.174
C08502=1232.266,369.180,-75.021,-175.795,7.387,148.174
C08503=1232.262,369.427,-75.054,-175.794,7.390,148.174
C08504=1232.258,369.675,-75.087,-175.793,7.393,148.175
C08505=1232.254,369.923,-75.120,-175.792,7.395,148.175
C08506=1232.250,370.171,-75.153,-175.790,7.398,148.175
C08507=1232.245,370.419,-75.186,-175.789,7.401,148.176
C08508=1232.241,370.666,-75.218,-175.788,7.404,148.176
C08509=1232.237,370.913,-75.251,-175.786,7.407,148.176
C08510=1232.233,371.162,-75.284,-175.785,7.408,148.176
C08511=1232.229,371.409,-75.317,-175.784,7.411,148.177
C08512=1232.225,371.657,-75.350,-175.783,7.414,148.177
C08513=1232.220,371.905,-75.383,-175.781,7.416,148.177
C08514=1232.216,372.153,-75.416,-175.780,7.419,148.178
C08515=1232.212,372.400,-75.450,-175.779,7.422,148.178
C08516=1232.208,372.649,-75.482,-175.777,7.425,148.178
C08517=1232.204,372.896,-75.515,-175.776,7.427,148.179
C08518=1232.199,373.144,-75.548,-175.775,7.430,148.179
C08519=1232.196,373.392,-75.581,-175.774,7.433,148.179
C08520=1232.192,373.639,-75.614,-175.773,7.435,148.180
C08521=1232.188,373.887,-75.647,-175.771,7.437,148.180
C08522=1232.184,374.135,-75.680,-175.770,7.440,148.180
C08523=1232.180,374.383,-75.713,-175.769,7.443,148.181
C08524=1232.175,374.630,-75.747,-175.767,7.445,148.181
C08525=1232.171,374.879,-75.779,-175.766,7.448,148.181
C08526=1232.167,375.126,-75.812,-175.765,7.451,148.182
C08527=1232.163,375.374,-75.845,-175.764,7.453,148.182
C08528=1232.159,375.622,-75.879,-175.763,7.456,148.182
C08529=1232.154,375.870,-75.912,-175.762,7.458,148.183
C08530=1232.150,376.117,-75.945,-175.760,7.461,148.183
C08531=1232.146,376.365,-75.978,-175.759,7.464,148.184
C08532=1232.142,376.613,-76.011,-175.758,7.467,148.184
C08533=1232.138,376.860,-76.044,-175.757,7.469,148.184
C08534=1232.134,377.108,-76.077,-175.756,7.471,148.184
C08535=1232.130,377.356,-76.111,-175.755,7.474,148.185
C08536=1232.125,377.604,-76.144,-175.753,7.477,148.185
C08537=1232.121,377.851,-76.177,-175.752,7.480,148.185
C08538=1232.118,378.100,-76.210,-175.751,7.482,148.186
C08539=1232.114,378.348,-76.244,-175.750,7.484,148.186
C08540=1232.109,378.595,-76.277,-175.749,7.487,148.187
C08541=1232.105,378.843,-76.310,-175.747,7.490,148.187
C08542=1232.102,379.090,-76.344,-175.746,7.493,148.187
C08543=1232.097,379.338,-76.377,-175.746,7.495,148.188
C08544=1232.092,379.586,-76.411,-175.744,7.497,148.188
C08545=1232.088,379.834,-76.444,-175.743,7.500,148.188
C08546=1232.084,380.081,-76.477,-175.742,7.503,148.189
C08547=1232.080,380.329,-76.510,-175.742,7.505,148.189
C08548=1232.076,380.577,-76.543,-175.740,7.508,148.189
C08549=1232.072,380.825,-76.577,-175.739,7.510,148.190
C08550=1232.068,381.072,-76.610,-175.738,7.513,148.190
C08551=1232.064,381.320,-76.643,-175.737,7.515,148.190
C08552=1232.060,381.567,-76.677,-175.736,7.518,148.191
C08553=1232.056,381.816,-76.710,-175.735,7.521,148.191
C08554=1232.051,382.064,-76.744,-175.734,7.524,148.192
C08555=1232.047,382.311,-76.777,-175.733,7.526,148.192
C08556=1232.043,382.559,-76.810,-175.731,7.528,148.192
C08557=1232.039,382.807,-76.843,-175.730,7.531,148.193
C08558=1232.035,383.054,-76.877,-175.729,7.533,148.193
C08559=1232.031,383.302,-76.910,-175.728,7.536,148.193
C08560=1232.027,383.549,-76.944,-175.727,7.539,148.194
C08561=1232.022,383.797,-76.977,-175.726,7.542,148.194
C08562=1232.018,384.044,-77.011,-175.725,7.543,148.194
C08563=1232.015,384.293,-77.045,-175.724,7.546,148.195
C08564=1232.010,384.541,-77.078,-175.723,7.549,148.195
C08565=1232.006,384.788,-77.111,-175.722,7.551,148.196
C08566=1232.002,385.035,-77.145,-175.721,7.554,148.196
C08567=1231.998,385.283,-77.179,-175.720,7.557,148.196
C08568=1231.993,385.531,-77.212,-175.719,7.559,148.197
C08569=1231.989,385.779,-77.245,-175.718,7.562,148.197
C08570=1231.985,386.026,-77.279,-175.717,7.564,148.198
C08571=1231.982,386.274,-77.312,-175.717,7.566,148.198
C08572=1231.977,386.523,-77.346,-175.715,7.569,148.198
C08573=1231.973,386.770,-77.380,-175.715,7.571,148.199
C08574=1231.969,387.017,-77.413,-175.714,7.574,148.199
C08575=1231.965,387.265,-77.446,-175.712,7.577,148.199
C08576=1231.961,387.512,-77.480,-175.712,7.579,148.200
C08577=1231.957,387.761,-77.514,-175.711,7.582,148.200
C08578=1231.953,388.009,-77.547,-175.709,7.584,148.201
C08579=1231.949,388.256,-77.581,-175.709,7.586,148.201
C08580=1231.945,388.504,-77.615,-175.708,7.589,148.201
C08581=1231.940,388.752,-77.648,-175.707,7.591,148.202
C08582=1231.936,388.999,-77.682,-175.706,7.594,148.202
C08583=1231.932,389.247,-77.716,-175.705,7.597,148.202
C08584=1231.929,389.494,-77.750,-175.704,7.599,148.203
C08585=1231.924,389.742,-77.783,-175.703,7.602,148.203
C08586=1231.920,389.990,-77.816,-175.702,7.604,148.204
C08587=1231.916,390.237,-77.850,-175.701,7.607,148.204
C08588=1231.911,390.485,-77.884,-175.701,7.609,148.204
C08589=1231.908,390.733,-77.918,-175.699,7.611,148.205
C08590=1231.904,390.981,-77.951,-175.698,7.614,148.205
C08591=1231.900,391.228,-77.985,-175.698,7.616,148.205
C08592=1231.895,391.476,-78.019,-175.696,7.619,148.206
C08593=1231.891,391.724,-78.052,-175.696,7.621,148.206
C08594=1231.887,391.971,-78.086,-175.695,7.624,148.207
C08595=1231.883,392.219,-78.120,-175.694,7.626,148.207
C08596=1231.879,392.466,-78.154,-175.693,7.629,148.208
C08597=1231.875,392.714,-78.187,-175.693,7.631,148.208
C08598=1231.870,392.996,-78.226,-175.692,7.634,148.208
C08599=1231.865,393.277,-78.264,-175.690,7.637,148.209
C08600=1231.861,393.558,-78.303,-175.690,7.640,148.209
C08601=1231.856,393.839,-78.342,-175.689,7.642,148.210
C08602=1231.852,394.087,-78.375,-175.688,7.644,148.210
C08603=1231.848,394.335,-78.409,-175.687,7.647,148.210
C08604=1231.844,394.583,-78.443,-175.686,7.649,148.211
C08605=1231.840,394.830,-78.477,-175.685,7.652,148.211
C08606=1231.836,395.077,-78.510,-175.685,7.654,148.212
C08607=1231.832,395.326,-78.545,-175.684,7.657,148.212
C08608=1231.827,395.573,-78.578,-175.683,7.659,148.212
C08609=1231.824,395.820,-78.612,-175.682,7.661,148.213
C08610=1231.819,396.068,-78.646,-175.681,7.664,148.213
C08611=1231.816,396.316,-78.680,-175.681,7.666,148.214
C08612=1231.811,396.564,-78.714,-175.679,7.669,148.214
C08613=1231.807,396.811,-78.747,-175.679,7.671,148.215
C08614=1231.803,397.059,-78.781,-175.678,7.674,148.215
C08615=1231.799,397.307,-78.816,-175.677,7.676,148.215
C08616=1231.795,397.554,-78.849,-175.676,7.679,148.216
C08617=1231.790,397.802,-78.884,-175.676,7.681,148.216
C08618=1231.786,398.049,-78.918,-175.675,7.683,148.216
C08619=1231.782,398.298,-78.952,-175.674,7.685,148.217
C08620=1231.778,398.545,-78.986,-175.674,7.688,148.217
C08621=1231.775,398.792,-79.020,-175.673,7.691,148.218
C08622=1231.770,399.041,-79.054,-175.672,7.693,148.218
C08623=1231.766,399.288,-79.088,-175.671,7.695,148.218
C08624=1231.762,399.535,-79.122,-175.670,7.697,148.219
C08625=1231.758,399.783,-79.155,-175.670,7.700,148.219
C08626=1231.754,400.031,-79.190,-175.669,7.702,148.220
C08627=1231.750,400.278,-79.224,-175.668,7.704,148.220
C08628=1231.745,400.526,-79.258,-175.668,7.706,148.220
C08629=1231.742,400.774,-79.292,-175.666,7.709,148.221
C08630=1231.738,401.021,-79.326,-175.666,7.711,148.221
C08631=1231.733,401.269,-79.359,-175.666,7.713,148.222
C08632=1231.729,401.516,-79.393,-175.664,7.716,148.222
C08633=1231.725,401.764,-79.428,-175.664,7.718,148.222
C08634=1231.721,402.011,-79.462,-175.663,7.721,148.223
C08635=1231.717,402.259,-79.496,-175.662,7.723,148.223
C08636=1231.713,402.507,-79.530,-175.662,7.725,148.224
C08637=1231.709,402.755,-79.564,-175.661,7.728,148.224
C08638=1231.705,403.002,-79.598,-175.660,7.730,148.224
C08639=1231.701,403.250,-79.633,-175.659,7.732,148.225
C08640=1231.697,403.498,-79.666,-175.659,7.734,148.225
C08641=1231.692,403.745,-79.701,-175.658,7.737,148.226
C08642=1231.689,403.993,-79.735,-175.657,7.739,148.226
C08643=1231.684,404.240,-79.769,-175.657,7.741,148.226
C08644=1231.680,404.488,-79.804,-175.656,7.744,148.227
C08645=1231.676,404.736,-79.837,-175.655,7.746,148.227
C08646=1231.672,404.984,-79.872,-175.655,7.748,148.228
C08647=1231.668,405.231,-79.906,-175.654,7.751,148.228
C08648=1231.664,405.479,-79.941,-175.653,7.753,148.228
C08649=1231.660,405.726,-79.975,-175.652,7.755,148.229
C08650=1231.656,405.973,-80.009,-175.652,7.757,148.229
C08651=1231.652,406.222,-80.043,-175.651,7.760,148.230
C08652=1231.648,406.469,-80.077,-175.650,7.762,148.230
C08653=1231.644,406.716,-80.111,-175.650,7.764,148.230
C08654=1231.640,406.964,-80.146,-175.649,7.767,148.231
C08655=1231.635,407.212,-80.180,-175.649,7.769,148.231
C08656=1231.631,407.459,-80.214,-175.648,7.771,148.232
C08657=1231.627,407.707,-80.249,-175.647,7.773,148.232
C08658=1231.624,407.954,-80.283,-175.646,7.776,148.233
C08659=1231.619,408.203,-80.317,-175.646,7.778,148.233
C08660=1231.615,408.450,-80.351,-175.645,7.780,148.233
C08661=1231.611,408.697,-80.385,-175.645,7.782,148.234
C08662=1231.607,408.946,-80.420,-175.644,7.784,148.234
C08663=1231.603,409.193,-80.454,-175.643,7.787,148.234
C08664=1231.598,409.440,-80.488,-175.643,7.789,148.235
C08665=1231.595,409.688,-80.523,-175.642,7.791,148.235
C08666=1231.591,409.935,-80.557,-175.641,7.793,148.236
C08667=1231.587,410.183,-80.592,-175.640,7.796,148.236
C08668=1231.583,410.431,-80.626,-175.640,7.798,148.237
C08669=1231.578,410.678,-80.660,-175.639,7.800,148.237
C08670=1231.574,410.926,-80.695,-175.639,7.802,148.237
C08671=1231.570,411.173,-80.729,-175.638,7.804,148.238
C08672=1231.567,411.421,-80.764,-175.637,7.807,148.238
C08673=1231.563,411.668,-80.798,-175.637,7.809,148.239
C08674=1231.558,411.916,-80.832,-175.636,7.811,148.239
C08675=1231.554,412.164,-80.867,-175.636,7.813,148.239
C08676=1231.550,412.411,-80.901,-175.635,7.815,148.240
C08677=1231.546,412.659,-80.936,-175.635,7.818,148.240
C08678=1231.542,412.907,-80.970,-175.634,7.820,148.241
C08679=1231.538,413.154,-81.004,-175.633,7.822,148.241
C08680=1231.534,413.402,-81.039,-175.632,7.824,148.241
C08681=1231.529,413.649,-81.073,-175.632,7.826,148.242
C08682=1231.526,413.897,-81.108,-175.632,7.829,148.242
C08683=1231.522,414.144,-81.142,-175.631,7.831,148.243
C08684=1231.517,414.392,-81.176,-175.630,7.833,148.243
C08685=1231.514,414.640,-81.211,-175.629,7.835,148.243
C08686=1231.509,414.887,-81.245,-175.629,7.838,148.244
C08687=1231.505,415.135,-81.280,-175.628,7.840,148.244
C08688=1231.501,415.382,-81.314,-175.628,7.842,148.244
C08689=1231.498,415.630,-81.349,-175.627,7.844,148.245
C08690=1231.491,415.997,-81.400,-175.626,7.847,148.245
C08691=1231.486,416.363,-81.451,-175.625,7.851,148.246
C08692=1231.479,416.730,-81.502,-175.624,7.854,148.247
C08693=1231.474,417.096,-81.553,-175.623,7.857,148.247
C08694=1231.051,417.096,-81.586,-175.627,7.867,148.251
C08695=1231.057,416.727,-81.534,-175.627,7.864,148.250
C08696=1231.063,416.358,-81.483,-175.629,7.860,148.250
C08697=1231.069,415.989,-81.432,-175.629,7.857,148.249
C08698=1231.075,415.620,-81.380,-175.631,7.854,148.249
C08699=1231.079,415.372,-81.345,-175.631,7.852,148.248
C08700=1231.083,415.125,-81.311,-175.631,7.850,148.248
C08701=1231.087,414.877,-81.276,-175.632,7.848,148.247
C08702=1231.092,414.629,-81.242,-175.633,7.846,148.247
C08703=1231.095,414.381,-81.207,-175.634,7.843,148.247
C08704=1231.100,414.134,-81.173,-175.634,7.841,148.246
C08705=1231.104,413.886,-81.138,-175.635,7.839,148.246
C08706=1231.107,413.639,-81.104,-175.635,7.837,148.245
C08707=1231.112,413.391,-81.070,-175.636,7.835,148.245
C08708=1231.116,413.143,-81.035,-175.636,7.833,148.245
C08709=1231.120,412.896,-81.001,-175.637,7.831,148.244
C08710=1231.124,412.649,-80.967,-175.638,7.828,148.244
C08711=1231.128,412.400,-80.932,-175.639,7.826,148.243
C08712=1231.132,412.153,-80.898,-175.639,7.824,148.243
C08713=1231.136,411.905,-80.863,-175.639,7.822,148.243
C08714=1231.141,411.658,-80.829,-175.640,7.820,148.242
C08715=1231.144,411.410,-80.794,-175.641,7.817,148.242
C08716=1231.149,411.163,-80.760,-175.642,7.815,148.241
C08717=1231.152,410.915,-80.726,-175.642,7.813,148.241
C08718=1231.156,410.667,-80.691,-175.643,7.811,148.241
C08719=1231.161,410.420,-80.657,-175.643,7.809,148.240
C08720=1231.164,410.172,-80.622,-175.644,7.806,148.240
C08721=1231.169,409.925,-80.588,-175.645,7.804,148.239
C08722=1231.173,409.677,-80.554,-175.645,7.802,148.239
C08723=1231.176,409.429,-80.519,-175.646,7.800,148.239
C08724=1231.181,409.182,-80.485,-175.646,7.798,148.238
C08725=1231.185,408.935,-80.451,-175.647,7.795,148.238
C08726=1231.189,408.687,-80.416,-175.648,7.793,148.237
C08727=1231.193,408.439,-80.382,-175.648,7.791,148.237
C08728=1231.197,408.192,-80.347,-175.649,7.789,148.237
C08729=1231.201,407.944,-80.313,-175.650,7.786,148.236
C08730=1231.205,407.697,-80.279,-175.650,7.784,148.236
C08731=1231.209,407.449,-80.244,-175.651,7.782,148.235
C08732=1231.214,407.202,-80.210,-175.652,7.780,148.235
C08733=1231.218,406.954,-80.177,-175.653,7.777,148.235
C08734=1231.222,406.706,-80.142,-175.653,7.774,148.234
C08735=1231.226,406.459,-80.108,-175.654,7.772,148.234
C08736=1231.230,406.211,-80.073,-175.654,7.771,148.233
C08737=1231.233,405.963,-80.039,-175.655,7.768,148.233
C08738=1231.238,405.716,-80.005,-175.656,7.765,148.232
C08739=1231.242,405.468,-79.970,-175.656,7.763,148.232
C08740=1231.246,405.221,-79.936,-175.657,7.761,148.232
C08741=1231.251,404.973,-79.902,-175.658,7.759,148.231
C08742=1231.254,404.725,-79.868,-175.659,7.757,148.231
C08743=1231.258,404.477,-79.834,-175.659,7.754,148.230
C08744=1231.262,404.230,-79.800,-175.660,7.752,148.230
C08745=1231.266,403.982,-79.765,-175.661,7.750,148.230
C08746=1231.270,403.735,-79.731,-175.661,7.748,148.229
C08747=1231.275,403.487,-79.697,-175.662,7.744,148.229
C08748=1231.278,403.239,-79.663,-175.663,7.742,148.228
C08749=1231.283,402.992,-79.629,-175.663,7.741,148.228
C08750=1231.287,402.745,-79.595,-175.664,7.738,148.228
C08751=1231.291,402.497,-79.561,-175.665,7.736,148.227
C08752=1231.295,402.249,-79.527,-175.665,7.733,148.227
C08753=1231.299,402.001,-79.492,-175.666,7.731,148.226
C08754=1231.303,401.754,-79.458,-175.667,7.729,148.226
C08755=1231.307,401.506,-79.424,-175.668,7.727,148.226
C08756=1231.311,401.258,-79.390,-175.669,7.724,148.225
C08757=1231.316,401.011,-79.356,-175.669,7.722,148.225
C08758=1231.319,400.763,-79.322,-175.670,7.720,148.224
C08759=1231.324,400.515,-79.288,-175.671,7.717,148.224
C08760=1231.328,400.268,-79.254,-175.671,7.715,148.224
C08761=1231.332,400.020,-79.219,-175.672,7.713,148.223
C08762=1231.335,399.773,-79.185,-175.673,7.710,148.223
C08763=1231.340,399.525,-79.152,-175.673,7.708,148.222
C08764=1231.344,399.278,-79.118,-175.674,7.705,148.222
C08765=1231.347,399.030,-79.084,-175.675,7.703,148.222
C08766=1231.352,398.782,-79.050,-175.676,7.701,148.221
C08767=1231.356,398.535,-79.016,-175.677,7.698,148.221
C08768=1231.361,398.287,-78.981,-175.677,7.696,148.220
C08769=1231.364,398.039,-78.948,-175.678,7.693,148.220
C08770=1231.369,397.791,-78.913,-175.679,7.691,148.220
C08771=1231.373,397.544,-78.880,-175.679,7.689,148.219
C08772=1231.377,397.296,-78.845,-175.681,7.686,148.219
C08773=1231.381,397.049,-78.812,-175.681,7.684,148.218
C08774=1231.385,396.801,-78.778,-175.682,7.681,148.218
C08775=1231.389,396.553,-78.744,-175.683,7.679,148.218
C08776=1231.393,396.306,-78.710,-175.684,7.676,148.217
C08777=1231.398,396.058,-78.676,-175.684,7.674,148.217
C08778=1231.401,395.810,-78.642,-175.686,7.671,148.216
C08779=1231.405,395.563,-78.608,-175.686,7.670,148.216
C08780=1231.409,395.315,-78.574,-175.687,7.666,148.215
C08781=1231.413,395.067,-78.540,-175.687,7.664,148.215
C08782=1231.417,394.820,-78.507,-175.688,7.662,148.215
C08783=1231.422,394.572,-78.473,-175.689,7.660,148.214
C08784=1231.426,394.324,-78.439,-175.690,7.658,148.214
C08785=1231.430,394.076,-78.405,-175.691,7.655,148.214
C08786=1231.434,393.829,-78.371,-175.692,7.653,148.213
C08787=1231.438,393.547,-78.333,-175.692,7.650,148.213
C08788=1231.443,393.267,-78.294,-175.694,7.647,148.212
C08789=1231.448,392.985,-78.256,-175.695,7.644,148.212
C08790=1231.452,392.704,-78.217,-175.696,7.641,148.211
C08791=1231.457,392.456,-78.184,-175.696,7.639,148.211
C08792=1231.461,392.209,-78.150,-175.697,7.636,148.211
C08793=1231.465,391.961,-78.116,-175.698,7.634,148.210
C08794=1231.469,391.713,-78.082,-175.699,7.631,148.210
C08795=1231.473,391.466,-78.049,-175.700,7.629,148.209
C08796=1231.477,391.218,-78.015,-175.701,7.627,148.209
C08797=1231.481,390.970,-77.981,-175.702,7.624,148.209
C08798=1231.486,390.722,-77.948,-175.703,7.622,148.208
C08799=1231.489,390.475,-77.914,-175.704,7.619,148.208
C08800=1231.493,390.227,-77.881,-175.704,7.617,148.208
C08801=1231.498,389.980,-77.846,-175.706,7.614,148.207
C08802=1231.502,389.732,-77.813,-175.706,7.612,148.207
C08803=1231.505,389.484,-77.779,-175.707,7.609,148.206
C08804=1231.510,389.236,-77.746,-175.708,7.606,148.206
C08805=1231.514,388.988,-77.712,-175.709,7.604,148.205
C08806=1231.518,388.741,-77.678,-175.710,7.601,148.205
C08807=1231.522,388.494,-77.645,-175.710,7.599,148.205
C08808=1231.526,388.246,-77.611,-175.712,7.597,148.204
C08809=1231.531,387.998,-77.577,-175.713,7.594,148.204
C08810=1231.535,387.750,-77.544,-175.713,7.592,148.204
C08811=1231.538,387.503,-77.510,-175.715,7.589,148.203
C08812=1231.543,387.255,-77.477,-175.715,7.587,148.203
C08813=1231.547,387.007,-77.443,-175.716,7.584,148.202
C08814=1231.551,386.759,-77.409,-175.717,7.581,148.202
C08815=1231.555,386.512,-77.375,-175.718,7.579,148.202
C08816=1231.559,386.264,-77.342,-175.719,7.576,148.201
C08817=1231.564,386.016,-77.308,-175.720,7.574,148.201
C08818=1231.568,385.769,-77.275,-175.721,7.572,148.201
C08819=1231.572,385.521,-77.242,-175.722,7.569,148.200
C08820=1231.576,385.273,-77.208,-175.723,7.566,148.200
C08821=1231.579,385.025,-77.174,-175.724,7.564,148.199
C08822=1231.583,384.778,-77.141,-175.725,7.561,148.199
C08823=1231.588,384.530,-77.107,-175.726,7.558,148.199
C08824=1231.592,384.283,-77.073,-175.727,7.556,148.198
C08825=1231.596,384.035,-77.040,-175.728,7.554,148.198
C08826=1231.600,383.787,-77.007,-175.729,7.551,148.197
C08827=1231.604,383.539,-76.974,-175.730,7.549,148.197
C08828=1231.609,383.291,-76.940,-175.731,7.546,148.197
C08829=1231.613,383.043,-76.906,-175.733,7.543,148.197
C08830=1231.617,382.796,-76.873,-175.733,7.541,148.196
C08831=1231.621,382.548,-76.840,-175.734,7.539,148.196
C08832=1231.625,382.300,-76.806,-175.736,7.536,148.195
C08833=1231.629,382.053,-76.773,-175.737,7.533,148.195
C08834=1231.633,381.805,-76.739,-175.737,7.531,148.195
C08835=1231.637,381.558,-76.706,-175.739,7.528,148.194
C08836=1231.642,381.310,-76.672,-175.740,7.525,148.194
C08837=1231.646,381.062,-76.639,-175.741,7.522,148.193
C08838=1231.650,380.814,-76.606,-175.742,7.521,148.193
C08839=1231.654,380.566,-76.573,-175.743,7.518,148.193
C08840=1231.658,380.319,-76.539,-175.744,7.515,148.192
C08841=1231.662,380.071,-76.506,-175.745,7.512,148.192
C08842=1231.666,379.823,-76.472,-175.746,7.510,148.192
C08843=1231.670,379.575,-76.439,-175.747,7.507,148.191
C08844=1231.674,379.328,-76.406,-175.748,7.505,148.191
C08845=1231.678,379.080,-76.373,-175.750,7.502,148.191
C08846=1231.682,378.832,-76.340,-175.751,7.500,148.190
C08847=1231.687,378.584,-76.306,-175.752,7.497,148.190
C08848=1231.691,378.337,-76.273,-175.753,7.494,148.190
C08849=1231.696,378.089,-76.240,-175.754,7.492,148.189
C08850=1231.700,377.841,-76.207,-175.755,7.489,148.189
C08851=1231.704,377.593,-76.173,-175.756,7.487,148.189
C08852=1231.708,377.346,-76.140,-175.758,7.484,148.188
C08853=1231.712,377.098,-76.107,-175.759,7.482,148.188
C08854=1231.716,376.850,-76.074,-175.760,7.479,148.187
C08855=1231.720,376.602,-76.041,-175.761,7.476,148.187
C08856=1231.725,376.355,-76.008,-175.762,7.474,148.187
C08857=1231.729,376.107,-75.975,-175.763,7.471,148.187
C08858=1231.733,375.859,-75.941,-175.764,7.469,148.186
C08859=1231.737,375.612,-75.908,-175.766,7.466,148.186
C08860=1231.741,375.364,-75.875,-175.767,7.463,148.186
C08861=1231.745,375.116,-75.842,-175.768,7.460,148.185
C08862=1231.749,374.868,-75.809,-175.769,7.457,148.185
C08863=1231.753,374.620,-75.775,-175.770,7.456,148.184
C08864=1231.757,374.372,-75.742,-175.772,7.453,148.184
C08865=1231.761,374.124,-75.709,-175.773,7.450,148.184
C08866=1231.765,373.877,-75.676,-175.774,7.447,148.183
C08867=1231.769,373.629,-75.643,-175.776,7.445,148.183
C08868=1231.774,373.381,-75.609,-175.777,7.442,148.183
C08869=1231.778,373.135,-75.577,-175.778,7.439,148.182
C08870=1231.782,372.887,-75.544,-175.780,7.437,148.182
C08871=1231.786,372.638,-75.512,-175.780,7.435,148.182
C08872=1231.790,372.391,-75.479,-175.781,7.432,148.181
C08873=1231.794,372.143,-75.445,-175.783,7.429,148.181
C08874=1231.799,371.895,-75.412,-175.784,7.426,148.181
C08875=1231.803,371.648,-75.379,-175.785,7.424,148.181
C08876=1231.807,371.400,-75.346,-175.787,7.421,148.180
C08877=1231.811,371.151,-75.313,-175.788,7.418,148.180
C08878=1231.815,370.904,-75.280,-175.790,7.416,148.180
C08879=1231.820,370.656,-75.247,-175.791,7.413,148.179
C08880=1231.823,370.409,-75.215,-175.792,7.410,148.179
C08881=1231.827,370.161,-75.181,-175.794,7.408,148.179
C08882=1231.832,369.912,-75.149,-175.795,7.405,148.178
C08883=1231.836,369.665,-75.116,-175.796,7.402,148.178
C08884=1231.840,369.417,-75.083,-175.798,7.399,148.178
C08885=1231.844,369.169,-75.050,-175.798,7.397,148.177
C08886=1231.848,368.921,-75.017,-175.800,7.395,148.177
C08887=1231.852,368.674,-74.985,-175.801,7.392,148.177
C08888=1231.856,368.426,-74.951,-175.803,7.389,148.177
C08889=1231.860,368.177,-74.919,-175.804,7.387,148.176
C08890=1231.865,367.930,-74.886,-175.805,7.384,148.176
C08891=1231.870,367.651,-74.849,-175.807,7.380,148.176
C08892=1231.874,367.372,-74.812,-175.809,7.378,148.175
C08893=1231.879,367.092,-74.775,-175.810,7.375,148.175
C08894=1231.884,366.813,-74.738,-175.812,7.371,148.175
C08895=1231.887,366.564,-74.706,-175.813,7.369,148.174
C08896=1231.892,366.317,-74.673,-175.815,7.366,148.174
C08897=1231.896,366.069,-74.640,-175.816,7.364,148.174
C08898=1231.900,365.821,-74.607,-175.818,7.361,148.174
C08899=1231.904,365.573,-74.575,-175.819,7.358,148.173
C08900=1231.908,365.326,-74.541,-175.820,7.356,148.173
C08901=1231.913,365.078,-74.509,-175.822,7.353,148.173
C08902=1231.917,364.830,-74.476,-175.823,7.350,148.172
C08903=1231.921,364.582,-74.444,-175.824,7.347,148.172
C08904=1231.925,364.334,-74.411,-175.826,7.345,148.172
C08905=1231.929,364.086,-74.379,-175.828,7.342,148.172
C08906=1231.933,363.838,-74.346,-175.829,7.340,148.171
C08907=1231.937,363.591,-74.313,-175.830,7.337,148.171
C08908=1231.941,363.343,-74.281,-175.832,7.334,148.171
C08909=1231.946,363.095,-74.248,-175.833,7.332,148.170
C08910=1231.950,362.847,-74.216,-175.835,7.329,148.170
C08911=1231.954,362.600,-74.183,-175.836,7.326,148.170
C08912=1231.958,362.351,-74.150,-175.838,7.324,148.170
C08913=1231.962,362.104,-74.118,-175.839,7.321,148.169
C08914=1231.966,361.856,-74.085,-175.840,7.318,148.169
C08915=1231.971,361.608,-74.053,-175.842,7.315,148.169
C08916=1231.974,361.361,-74.021,-175.844,7.313,148.169
C08917=1231.979,361.112,-73.988,-175.845,7.310,148.168
C08918=1231.983,360.864,-73.955,-175.847,7.307,148.168
C08919=1231.987,360.616,-73.923,-175.849,7.305,148.168
C08920=1231.991,360.369,-73.890,-175.850,7.302,148.168
C08921=1231.996,360.121,-73.858,-175.851,7.299,148.167
C08922=1232.000,359.873,-73.826,-175.853,7.297,148.167
C08923=1232.004,359.625,-73.793,-175.855,7.294,148.167
C08924=1232.008,359.377,-73.761,-175.856,7.292,148.167
C08925=1232.012,359.130,-73.728,-175.857,7.289,148.166
C08926=1232.017,358.882,-73.696,-175.859,7.286,148.166
C08927=1232.020,358.634,-73.664,-175.861,7.283,148.166
C08928=1232.025,358.386,-73.631,-175.863,7.280,148.166
C08929=1232.029,358.138,-73.598,-175.864,7.278,148.165
C08930=1232.033,357.890,-73.567,-175.866,7.275,148.165
C08931=1232.037,357.643,-73.534,-175.867,7.273,148.165
C08932=1232.041,357.395,-73.502,-175.869,7.270,148.165
C08933=1232.046,357.146,-73.470,-175.870,7.267,148.165
C08934=1232.049,356.898,-73.438,-175.872,7.265,148.164
C08935=1232.054,356.651,-73.405,-175.873,7.262,148.164
C08936=1232.058,356.403,-73.373,-175.875,7.260,148.164
C08937=1232.062,356.155,-73.341,-175.877,7.256,148.164
C08938=1232.066,355.907,-73.309,-175.879,7.254,148.163
C08939=1232.071,355.660,-73.276,-175.880,7.251,148.163
C08940=1232.075,355.411,-73.244,-175.882,7.249,148.163
C08941=1232.079,355.163,-73.212,-175.883,7.246,148.163
C08942=1232.083,354.915,-73.179,-175.885,7.243,148.162
C08943=1232.087,354.668,-73.147,-175.886,7.241,148.162
C08944=1232.092,354.420,-73.115,-175.888,7.238,148.162
C08945=1232.095,354.172,-73.083,-175.890,7.235,148.162
C08946=1232.100,353.925,-73.051,-175.892,7.232,148.162
C08947=1232.104,353.676,-73.019,-175.893,7.230,148.161
C08948=1232.108,353.428,-72.987,-175.895,7.227,148.161
C08949=1232.112,353.180,-72.955,-175.896,7.225,148.161
C08950=1232.116,352.933,-72.922,-175.898,7.222,148.161
C08951=1232.121,352.685,-72.890,-175.900,7.220,148.161
C08952=1232.124,352.437,-72.858,-175.902,7.216,148.160
C08953=1232.129,352.189,-72.826,-175.903,7.213,148.160
C08954=1232.133,351.941,-72.794,-175.905,7.211,148.160
C08955=1232.138,351.693,-72.762,-175.906,7.208,148.160
C08956=1232.142,351.445,-72.730,-175.908,7.206,148.160
C08957=1232.146,351.197,-72.698,-175.910,7.203,148.159
C08958=1232.150,350.949,-72.666,-175.912,7.200,148.159
C08959=1232.154,350.702,-72.635,-175.913,7.197,148.159
C08960=1232.159,350.453,-72.602,-175.915,7.195,148.159
C08961=1232.163,350.205,-72.570,-175.917,7.192,148.159
C08962=1232.167,349.958,-72.539,-175.918,7.190,148.158
C08963=1232.171,349.710,-72.506,-175.920,7.188,148.158
C08964=1232.175,349.462,-72.474,-175.922,7.184,148.158
C08965=1232.179,349.214,-72.443,-175.924,7.182,148.158
C08966=1232.184,348.966,-72.411,-175.926,7.179,148.158
C08967=1232.187,348.718,-72.379,-175.927,7.177,148.158
C08968=1232.192,348.470,-72.347,-175.929,7.174,148.157
C08969=1232.196,348.222,-72.315,-175.931,7.171,148.157
C08970=1232.200,347.974,-72.283,-175.933,7.168,148.157
C08971=1232.204,347.727,-72.251,-175.934,7.166,148.157
C08972=1232.209,347.478,-72.219,-175.936,7.163,148.157
C08973=1232.213,347.230,-72.188,-175.938,7.161,148.156
C08974=1232.217,346.982,-72.156,-175.939,7.158,148.156
C08975=1232.221,346.734,-72.124,-175.942,7.155,148.156
C08976=1232.226,346.487,-72.092,-175.943,7.152,148.156
C08977=1232.229,346.239,-72.061,-175.945,7.150,148.156
C08978=1232.234,345.991,-72.029,-175.947,7.147,148.156
C08979=1232.238,345.743,-71.997,-175.948,7.145,148.156
C08980=1232.242,345.494,-71.966,-175.950,7.141,148.155
C08981=1232.246,345.247,-71.934,-175.952,7.139,148.155
C08982=1232.250,344.999,-71.902,-175.954,7.137,148.155
C08983=1232.255,344.751,-71.870,-175.956,7.134,148.155
C08984=1232.259,344.503,-71.838,-175.957,7.132,148.155
C08985=1232.263,344.255,-71.807,-175.960,7.128,148.155
C08986=1232.267,344.007,-71.776,-175.961,7.126,148.154
C08987=1232.272,343.759,-71.743,-175.963,7.123,148.154
C08988=1232.276,343.512,-71.712,-175.965,7.121,148.154
C08989=1232.280,343.263,-71.681,-175.967,7.118,148.154
C08990=1232.284,343.016,-71.649,-175.969,7.115,148.154
C08991=1232.288,342.768,-71.617,-175.970,7.112,148.154
C08992=1232.293,342.519,-71.586,-175.972,7.110,148.154
C08993=1232.297,342.271,-71.554,-175.974,7.108,148.154
C08994=1232.301,342.024,-71.523,-175.976,7.105,148.153
C08995=1232.306,341.746,-71.488,-175.978,7.102,148.153
C08996=1232.310,341.468,-71.452,-175.981,7.099,148.153
C08997=1232.315,341.191,-71.417,-175.982,7.096,148.153
C08998=1232.320,340.913,-71.382,-175.984,7.093,148.153
C08999=1232.324,340.666,-71.351,-175.986,7.091,148.153
C09000=1232.329,340.417,-71.319,-175.988,7.088,148.153
C09001=1232.333,340.170,-71.287,-175.990,7.086,148.152
C09002=1232.337,339.922,-71.256,-175.992,7.082,148.152
C09003=1232.342,339.674,-71.225,-175.994,7.080,148.152
C09004=1232.345,339.426,-71.193,-175.996,7.077,148.152
C09005=1232.350,339.178,-71.162,-175.997,7.075,148.152
C09006=1232.354,338.930,-71.130,-176.000,7.072,148.152
C09007=1232.358,338.682,-71.100,-176.001,7.069,148.152
C09008=1232.362,338.434,-71.068,-176.003,7.067,148.151
C09009=1232.367,338.186,-71.037,-176.005,7.064,148.151
C09010=1232.370,337.938,-71.005,-176.007,7.062,148.151
C09011=1232.375,337.690,-70.974,-176.009,7.059,148.151
C09012=1232.379,337.442,-70.942,-176.011,7.056,148.151
C09013=1232.383,337.194,-70.912,-176.013,7.054,148.151
C09014=1232.388,336.945,-70.879,-176.015,7.052,148.151
C09015=1232.392,336.697,-70.849,-176.017,7.048,148.151
C09016=1232.396,336.449,-70.817,-176.018,7.046,148.150
C09017=1232.401,336.201,-70.786,-176.021,7.043,148.151
C09018=1232.405,335.953,-70.755,-176.022,7.041,148.150
C09019=1232.409,335.705,-70.723,-176.025,7.038,148.150
C09020=1232.413,335.457,-70.693,-176.026,7.035,148.150
C09021=1232.416,335.210,-70.661,-176.029,7.033,148.150
C09022=1232.421,334.962,-70.631,-176.030,7.031,148.150
C09023=1232.425,334.713,-70.599,-176.032,7.027,148.150
C09024=1232.429,334.466,-70.568,-176.034,7.025,148.150
C09025=1232.434,334.218,-70.537,-176.036,7.022,148.150
C09026=1232.438,333.969,-70.506,-176.038,7.020,148.150
C09027=1232.442,333.722,-70.475,-176.040,7.018,148.150
C09028=1232.446,333.473,-70.443,-176.042,7.015,148.149
C09029=1232.451,333.225,-70.413,-176.044,7.012,148.149
C09030=1232.455,332.978,-70.381,-176.046,7.010,148.149
C09031=1232.459,332.729,-70.350,-176.048,7.007,148.149
C09032=1232.464,332.481,-70.319,-176.050,7.004,148.149
C09033=1232.468,332.232,-70.288,-176.052,7.002,148.149
C09034=1232.472,331.985,-70.257,-176.054,6.999,148.149
C09035=1232.476,331.738,-70.226,-176.056,6.997,148.149
C09036=1232.480,331.489,-70.195,-176.058,6.994,148.149
C09037=1232.485,331.241,-70.165,-176.060,6.991,148.149
C09038=1232.489,330.993,-70.134,-176.062,6.989,148.149
C09039=1232.493,330.745,-70.102,-176.064,6.987,148.149
C09040=1232.498,330.497,-70.071,-176.066,6.983,148.149
C09041=1232.502,330.249,-70.040,-176.068,6.981,148.148
C09042=1232.506,330.001,-70.010,-176.070,6.979,148.148
C09043=1232.510,329.753,-69.979,-176.072,6.977,148.148
C09044=1232.515,329.505,-69.948,-176.074,6.973,148.148
C09045=1232.519,329.256,-69.917,-176.076,6.971,148.148
C09046=1232.523,329.009,-69.886,-176.078,6.968,148.148
C09047=1232.528,328.761,-69.855,-176.080,6.966,148.148
C09048=1232.531,328.512,-69.824,-176.082,6.963,148.148
C09049=1232.536,328.264,-69.794,-176.084,6.961,148.148
C09050=1232.540,328.016,-69.763,-176.087,6.958,148.148
C09051=1232.544,327.768,-69.732,-176.088,6.956,148.148
C09052=1232.548,327.520,-69.702,-176.091,6.953,148.148
C09053=1232.553,327.272,-69.671,-176.093,6.950,148.148
C09054=1232.557,327.024,-69.640,-176.094,6.948,148.148
C09055=1232.561,326.776,-69.609,-176.097,6.946,148.148
C09056=1232.565,326.528,-69.579,-176.099,6.942,148.147
C09057=1232.570,326.280,-69.548,-176.101,6.940,148.147
C09058=1232.574,326.031,-69.517,-176.103,6.938,148.148
C09059=1232.578,325.784,-69.487,-176.105,6.935,148.147
C09060=1232.582,325.536,-69.456,-176.107,6.932,148.147
C09061=1232.587,325.288,-69.425,-176.109,6.930,148.147
C09062=1232.591,325.039,-69.394,-176.111,6.928,148.147
C09063=1232.595,324.791,-69.364,-176.113,6.925,148.147
C09064=1232.599,324.544,-69.333,-176.116,6.922,148.147
C09065=1232.604,324.296,-69.302,-176.117,6.920,148.147
C09066=1232.607,324.047,-69.272,-176.119,6.917,148.147
C09067=1232.612,323.799,-69.242,-176.121,6.915,148.147
C09068=1232.617,323.551,-69.211,-176.124,6.912,148.147
C09069=1232.621,323.303,-69.181,-176.126,6.910,148.147
C09070=1232.625,323.054,-69.150,-176.128,6.907,148.147
C09071=1232.629,322.807,-69.120,-176.130,6.905,148.147
C09072=1232.633,322.559,-69.089,-176.132,6.902,148.147
C09073=1232.638,322.310,-69.059,-176.134,6.900,148.147
C09074=1232.642,322.063,-69.029,-176.136,6.897,148.147
C09075=1232.646,321.814,-68.997,-176.139,6.894,148.147
C09076=1232.650,321.566,-68.967,-176.141,6.892,148.147
C09077=1232.655,321.318,-68.937,-176.143,6.890,148.147
C09078=1232.659,321.070,-68.907,-176.145,6.887,148.147
C09079=1232.663,320.822,-68.876,-176.147,6.884,148.147
C09080=1232.667,320.573,-68.845,-176.149,6.882,148.147
C09081=1232.671,320.326,-68.815,-176.151,6.879,148.147
C09082=1232.676,320.077,-68.785,-176.153,6.877,148.147
C09083=1232.680,319.830,-68.755,-176.156,6.874,148.147
C09084=1232.685,319.582,-68.724,-176.158,6.872,148.147
C09085=1232.689,319.333,-68.695,-176.160,6.869,148.147
C09086=1232.693,319.085,-68.663,-176.162,6.867,148.147
C09087=1232.697,318.837,-68.633,-176.164,6.864,148.147
C09088=1232.702,318.588,-68.603,-176.166,6.862,148.147
C09089=1232.706,318.340,-68.572,-176.169,6.860,148.147
C09090=1232.710,318.093,-68.542,-176.171,6.857,148.147
C09091=1232.714,317.845,-68.513,-176.173,6.854,148.147
C09092=1232.719,317.597,-68.482,-176.175,6.852,148.147
C09093=1232.722,317.348,-68.452,-176.177,6.850,148.147
C09094=1232.727,317.100,-68.422,-176.179,6.847,148.147
C09095=1232.731,316.852,-68.391,-176.182,6.844,148.147
C09096=1232.736,316.603,-68.361,-176.184,6.842,148.147
C09097=1232.740,316.356,-68.331,-176.185,6.840,148.147
C09098=1232.745,316.107,-68.301,-176.188,6.837,148.147
C09099=1232.749,315.832,-68.267,-176.190,6.834,148.147
C09100=1232.754,315.556,-68.234,-176.193,6.831,148.147
C09101=1232.758,315.281,-68.201,-176.195,6.829,148.147
C09102=1232.763,315.004,-68.168,-176.198,6.826,148.147
C09103=1232.767,314.756,-68.137,-176.200,6.824,148.147
C09104=1232.772,314.508,-68.107,-176.202,6.821,148.147
C09105=1232.776,314.260,-68.077,-176.204,6.818,148.147
C09106=1232.780,314.012,-68.047,-176.206,6.816,148.147
C09107=1232.785,313.764,-68.018,-176.209,6.814,148.147
C09108=1232.789,313.516,-67.987,-176.211,6.812,148.147
C09109=1232.793,313.268,-67.957,-176.213,6.809,148.147
C09110=1232.797,313.020,-67.927,-176.215,6.806,148.147
C09111=1232.802,312.771,-67.897,-176.218,6.804,148.147
C09112=1232.806,312.523,-67.868,-176.220,6.802,148.147
C09113=1232.810,312.275,-67.838,-176.221,6.799,148.147
C09114=1232.815,312.027,-67.808,-176.224,6.796,148.147
C09115=1232.819,311.779,-67.777,-176.226,6.794,148.147
C09116=1232.823,311.531,-67.748,-176.228,6.792,148.147
C09117=1232.828,311.282,-67.718,-176.230,6.790,148.147
C09118=1232.832,311.034,-67.688,-176.233,6.787,148.147
C09119=1232.836,310.786,-67.658,-176.235,6.784,148.147
C09120=1232.840,310.537,-67.628,-176.237,6.782,148.147
C09121=1232.845,310.289,-67.598,-176.239,6.780,148.147
C09122=1232.849,310.041,-67.568,-176.242,6.777,148.147
C09123=1232.853,309.793,-67.539,-176.244,6.775,148.147
C09124=1232.858,309.545,-67.509,-176.246,6.772,148.147
